# B&R Automation Studio project Template
Automation Studio 4.9

## Logical view

### axisConfiguration.typ - Global data types
```iecst
TYPE
	global_command_typ : 	STRUCT  (*command structure for global commands*)
		Power : BOOL; (*switch on the controller of all axes*)
		Home : BOOL; (*reference all axes*)
		Stop : BOOL; (*stop everey active movement as long as is set (emergency stop)*)
		ErrorAcknowledge : BOOL; (*reset active errors*)
	END_STRUCT;
	psm_command_typ : 	STRUCT  (*command structure for power supply modules*)
		Power : BOOL; (*switch on the controller of the psm*)
		StartPowerMeter : BOOL; (*start the power evaluation of psm*)
		StopPowerMeter : BOOL; (*stop the power evaluation of psm*)
		RestartInterval : BOOL; (*restart the interval of power evaluation*)
	END_STRUCT;
	axis_command_typ : 	STRUCT  (*command structure for single and master axes*)
		Power : BOOL; (*switch on the controller*)
		Home : BOOL; (*reference axis*)
		MoveJogPos : BOOL; (*move in positive direction as long as is set*)
		MoveJogNeg : BOOL; (*move in negative direction as long as is set*)
		MoveAbsolute : BOOL; (*move to a defined position*)
		MoveAdditive : BOOL; (*move a defined distance*)
		MoveVelocity : BOOL; (*start a movement with a defined velocity*)
		Stop : BOOL; (*stop every active movement on the axis as long as is set*)
		Halt : BOOL; (*stop every active movement on the axis*)
	END_STRUCT;
	slave_command_typ : 	STRUCT  (*command structure for slave axes*)
		Power : BOOL; (*switch on the controller*)
		Home : BOOL; (*reference axis*)
		MoveJogPos : BOOL; (*move in positive direction as long as is set*)
		MoveJogNeg : BOOL; (*move in negative direction as long as is set*)
		MoveAbsolute : BOOL; (*move to a defined position*)
		MoveAdditive : BOOL; (*move a defined distance*)
		MoveVelocity : BOOL; (*start a movement with a defined velocity*)
		Stop : BOOL; (*stop every active movement on the axis as long as is set*)
		Halt : BOOL; (*stop every active movement on the axis*)
		StartAutomat : BOOL; (*start coupling between master and slave*)
		StopSlave : BOOL; (*stop coupling between master and slave (automat is still active)*)
		RestartAutomat : BOOL; (*reengage the coupling between master and slave*)
		EndAutomat : BOOL; (*terminate the automat*)
		SetSignal1 : BOOL; (*set the first signal of the automat*)
		SetSignal2 : BOOL; (*set the second signal of the automat*)
		SetSignal3 : BOOL; (*set the third signal of the automat*)
		SetSignal4 : BOOL; (*set the fourth signal of the automat*)
		ResetSignal1 : BOOL; (*reset the first signal of the automat*)
		ResetSignal2 : BOOL; (*reset the second signal of the automat*)
		ResetSignal3 : BOOL; (*reset the third signal of the automat*)
		ResetSignal4 : BOOL; (*reset the fourth signal of the automat*)
	END_STRUCT;
	parameter_typ : 	STRUCT  (*parameter structure*)
		Position : REAL; (*target position for MoveAbsolute-Command*)
		Distance : REAL; (*distance for MoveAdditive-Command*)
		Velocity : REAL; (*velocity for MoveVelocity-Command*)
		Direction : USINT; (*direction for commanded movements*)
		Acceleration : REAL; (*acceleration for commanded movements*)
		Deceleration : REAL; (*deceleration for commanded movements*)
		HomePosition : REAL; (*target position for referencing the axis*)
		HomeMode : USINT; (*homing mode*)
		JogVelocity : REAL; (*velocity for jogging movement*)
	END_STRUCT;
	psm_parameter_typ : 	STRUCT  (*parameter structure for psm*)
		IntervalTime : UINT; (*interval time for the power evaluation*)
	END_STRUCT;
	status_typ : 	STRUCT  (*status structure*)
		ActPosition : REAL; (*actual position of the axis*)
		ActVelocity : REAL; (*actual velocity of the axis*)
		DriveStatus : MC_DRIVESTATUS_TYP; (*actual status of the axis*)
	END_STRUCT;
	slave_status_typ : 	STRUCT  (*status structure*)
		ActPosition : REAL; (*actual position of the axis*)
		ActVelocity : REAL; (*actual velocity of the axis*)
		AutomatRunning : BOOL; (*if set, automat is running*)
		AutomatStandBy : BOOL; (*if set, automat is in stand by*)
		ActualStateIndex : USINT; (*actual state index of the cam automat*)
		ActualStateCamIndex : UINT; (*actual index of the cam profile*)
		InCam : BOOL; (*if set, the cam profile is active*)
		InCompensation : BOOL; (*if set, compensation is active*)
		DriveStatus : MC_DRIVESTATUS_TYP; (*actual status of the axis*)
	END_STRUCT;
	psm_status_typ : 	STRUCT  (*status structure for psm*)
		PowerData : MC_POWERDATA_REF; (*evaluated power data*)
		MissedInterval : UINT; (*MissedIntervals with power evaluation*)
		DriveStatus : MC_DRIVESTATUS_TYP; (*actual status of the axis*)
	END_STRUCT;
	axisState_typ : 	STRUCT  (*axis state structure*)
		Disabled : BOOL; (*if set, axis is in state Disabled*)
		StandStill : BOOL; (*if set, axis is in state StandsStill*)
		Homing : BOOL; (*if set, axis is in state Homing*)
		Stopping : BOOL; (*if set, axis is in state Stopping*)
		DiscreteMotion : BOOL; (*if set, axis is in state DiscreteMotion*)
		ContinuousMotion : BOOL; (*if set, axis is in state ContinuousMotion*)
		SynchronizedMotion : BOOL; (*if set, axis is in state SynchronizedMotion*)
		ErrorStop : BOOL; (*if set, axis is in state ErrorStop*)
	END_STRUCT;
	error_typ : 	STRUCT  (*error structure *)
		AxisErrorCount : UINT; (*number of active axis errors*)
		AxisWarningCount : UINT; (*number of active axis warinings*)
		FunctionBlockErrorCount : UINT; (*number of active function block errors*)
		ErrorRecord : MC_ERRORRECORD_REF; (*error record information*)
		ErrorText : ARRAY[0..3] OF STRING[79]; (*description of first active error or warning*)
	END_STRUCT;
	axis_typ : 	STRUCT  (*substructure for single and master axes*)
		Command : axis_command_typ; (*command structure for single and master axes*)
		Parameter : parameter_typ; (*parameter structure*)
		Status : status_typ; (*status structure*)
		AxisState : axisState_typ; (*axis state structure*)
		Error : error_typ; (*error structure*)
	END_STRUCT;
	slave_typ : 	STRUCT  (*substructure for slave axis*)
		Command : slave_command_typ; (*command structure for slave axes*)
		Parameter : parameter_typ; (*parameter structure*)
		Status : slave_status_typ; (*status structure*)
		AxisState : axisState_typ; (*axis state structure*)
		Error : error_typ; (*error structure*)
	END_STRUCT;
	psm_typ : 	STRUCT  (*substructure for psm*)
		Command : psm_command_typ; (*command structure for psm*)
		Parameter : psm_parameter_typ; (*parameter structure for psm*)
		Status : psm_status_typ; (*status structure for psm*)
		AxisState : axisState_typ; (*axis state structure*)
		Error : error_typ; (*error structure*)
	END_STRUCT;
	global_error_typ : 	STRUCT  (*error structure for global errors*)
		AxisTyp : STRING[10]; (*axis type (Axis, Master or Slave)*)
		AxisIndex : USINT; (*index of error reporting axis (total axis index)*)
		ErrorText : ARRAY[0..3] OF STRING[79]; (*description of first active error or warning*)
		ErrorRecord : MC_ERRORRECORD_REF; (*error record information*)
	END_STRUCT;
END_TYPE
```

### axisConfiguration.var - Global variables
```iecst
VAR CONSTANT
	PSM_NUMBER : USINT := 1; (*number of used power supply modules*)
	AXIS_NUMBER : USINT := 2; (*number of used single axes*)
	MASTER_NUMBER : USINT := 1; (*number of used master axes*)
	SLAVE_NUMBER : USINT := 1; (*number of used slave axes*)
	TOTAL_AXES : USINT := PSM_NUMBER + AXIS_NUMBER + MASTER_NUMBER + SLAVE_NUMBER; (*total number of used axes*)
	PSM_MAX_INDEX : USINT := PSM_NUMBER-1; (*highest index for single axis*)
	AXIS_MAX_INDEX : USINT := AXIS_NUMBER-1; (*highest index for single axes*)
	MASTER_MAX_INDEX : USINT := MASTER_NUMBER-1; (*highest index for master axes*)
	SLAVE_MAX_INDEX : USINT := SLAVE_NUMBER-1; (*highest index for slave axes*)
END_VAR
VAR
	PsmRef : ARRAY[0..PSM_MAX_INDEX] OF UDINT; (*psm reference handle*)
	AxisRef : ARRAY[0..AXIS_MAX_INDEX] OF UDINT; (*axis reference handle*)
	MasterRef : ARRAY[0..MASTER_MAX_INDEX] OF UDINT; (*master reference handle*)
	SlaveRef : ARRAY[0..SLAVE_MAX_INDEX] OF UDINT; (*slave reference handle*)
	GlobalCommand : global_command_typ; (*command structure for global command*)
	GlobalError : global_error_typ; (*error structure for global error*)
	PowerSupply : ARRAY[0..PSM_MAX_INDEX] OF psm_typ; (*handling structure for power supply module*)
	Axis : ARRAY[0..AXIS_MAX_INDEX] OF axis_typ; (*handling structure for single axis*)
	Master : ARRAY[0..MASTER_MAX_INDEX] OF axis_typ; (*handling structure for master axis*)
	Slave : ARRAY[0..SLAVE_MAX_INDEX] OF slave_typ; (*handling structure for slave axis*)
	PowerSupplyOn : BOOL; (*power supply on flag*)
END_VAR
```

### Program Logical/LibACP10MC_MotionControl_ST/AxisConfiguration (IEC) - configuration task

#### axisConfiguration.st - Implementation code
```iecst
(********************************************************************
 * COPYRIGHT -- Bernecker + Rainer
 ********************************************************************
 * Program: AxisConfiguration
 * File: axisConfiguration.st
 * Author: Bernecker + Rainer
 * Created: March 01, 2011
 ********************************************************************
 * Implementation of program AxisConfiguration
 ********************************************************************)

PROGRAM _INIT
    PsmRef[0] := ADR(gAxis01); (* axis reference of the power supply module *)
    AxisRef[0] := ADR(gAxis02); (* axis reference of first single axis *)
    AxisRef[1] := ADR(gAxis03); (* axis reference of second single axis *)
    MasterRef[0] := ADR(gAxis04); (* axis reference of first master axis *)
    SlaveRef[0] := ADR(gAxis05); (* axis reference of first slave axis *)

    PowerSupplyOn := TRUE; (* if a power supply is used, this variable is reset in the according task *)
END_PROGRAM
```

### Program Logical/LibACP10MC_MotionControl_ST/PowerSupply (IEC) - power supply handle

#### powerSupplyCyclic.st - Cyclic code
```iecst
(********************************************************************
 * COPYRIGHT -- Bernecker + Rainer
 ********************************************************************
 * Program: PowerSupply
 * File: powerSupplyCyclic.st
 * Author: Bernecker + Rainer
 * Created: March 01, 2011
 ********************************************************************
 * Implementation of program PowerSupply
 ********************************************************************)

PROGRAM _CYCLIC

(************************** MC_READSTATUS ***************************)
MC_ReadStatus_0.Enable := NOT(MC_ReadStatus_0.Error);
MC_ReadStatus_0.Axis := PsmRef[PSM_INDEX];
MC_ReadStatus_0();
PowerSupply[PSM_INDEX].AxisState.Disabled := MC_ReadStatus_0.Disabled;
PowerSupply[PSM_INDEX].AxisState.StandStill := MC_ReadStatus_0.StandStill;
PowerSupply[PSM_INDEX].AxisState.Stopping := MC_ReadStatus_0.Stopping;
PowerSupply[PSM_INDEX].AxisState.Homing := MC_ReadStatus_0.Homing;
PowerSupply[PSM_INDEX].AxisState.DiscreteMotion := MC_ReadStatus_0.DiscreteMotion;
PowerSupply[PSM_INDEX].AxisState.ContinuousMotion := MC_ReadStatus_0.ContinuousMotion;
PowerSupply[PSM_INDEX].AxisState.SynchronizedMotion := MC_ReadStatus_0.SynchronizedMotion;
PowerSupply[PSM_INDEX].AxisState.ErrorStop := MC_ReadStatus_0.Errorstop;

(************************* MC_BR_READDRIVESTATUS ********************)
MC_BR_ReadDriveStatus_0.Enable := NOT(MC_BR_ReadDriveStatus_0.Error);
MC_BR_ReadDriveStatus_0.Axis := PsmRef[PSM_INDEX];
MC_BR_ReadDriveStatus_0.AdrDriveStatus := ADR(PowerSupply[PSM_INDEX].Status.DriveStatus);
MC_BR_ReadDriveStatus_0();

CASE PsmStep OF
(********************************* READY ****************************)
    STATE_READY:
        IF (((GlobalCommand.Power = TRUE) OR (PowerSupply[PSM_INDEX].Command.Power = TRUE)) AND
             (MC_Power_0.Status = FALSE)) THEN
            PsmStep := STATE_POWER_ON;
        ELSIF ((GlobalCommand.Power = FALSE) AND (PowerSupply[PSM_INDEX].Command.Power = FALSE) AND
                 (MC_Power_0.Status = TRUE)) THEN
            PsmStep := STATE_POWER_OFF;
        ELSIF (PowerSupply[PSM_INDEX].Command.StartPowerMeter = TRUE) THEN
            PowerSupply[PSM_INDEX].Command.StartPowerMeter := FALSE;
            PsmStep := STATE_START_POWERMETER;
        ELSIF (PowerSupply[PSM_INDEX].Command.StopPowerMeter = TRUE) THEN
            PowerSupply[PSM_INDEX].Command.StopPowerMeter := FALSE;
            PsmStep := STATE_STOP_POWERMETER;
        ELSIF (PowerSupply[PSM_INDEX].Command.RestartInterval = TRUE) THEN
            PowerSupply[PSM_INDEX].Command.RestartInterval := FALSE;
            MC_BR_PowerMeter_0.RestartInterval := FALSE;
            PsmStep := STATE_RESTART_INTERVAL;
        END_IF

        (* End of STATE_READY *)

(*************************** POWER ON ********************************)
    STATE_POWER_ON:
        MC_Power_0.Enable := TRUE;
        IF (MC_Power_0.Status = TRUE) THEN
            PsmStep := STATE_READY;
        END_IF

        (* IF a power error occured switch off controller *)
        IF (MC_Power_0.Error = TRUE) THEN
            MC_Power_0.Enable := FALSE;
        END_IF

        (* End of STATE_POWER_ON *)

(************************* POWER OFF *******************************)
    STATE_POWER_OFF:
        MC_Power_0.Enable := FALSE;
        IF (MC_Power_0.Status = FALSE) THEN
            PsmStep := STATE_READY;
        END_IF

        (* End of STATE_POWER_OFF *)

(************************ START POWERMETER **************************)
    STATE_START_POWERMETER:
        MC_BR_PowerMeter_0.Enable := TRUE;
        MC_BR_PowerMeter_0.Mode := mcONLY_PSM;
        MC_BR_PowerMeter_0.IntervalTime := PowerSupply[PSM_INDEX].Parameter.IntervalTime;

        IF (MC_BR_PowerMeter_0.Valid = TRUE) THEN
            PsmStep := STATE_READY;
        END_IF

        (* check IF error occured *)
        IF (MC_BR_PowerMeter_0.Error = TRUE) THEN
            MC_BR_PowerMeter_0.Enable := FALSE;
            PsmStep := STATE_READY;
        END_IF

        (* End of STATE_START_POWERMETER *)

(************************ STOP POWERMETER ***************************)
    STATE_STOP_POWERMETER:
        MC_BR_PowerMeter_0.Enable := FALSE;

        IF (MC_BR_PowerMeter_0.Valid = FALSE) THEN
            PsmStep := STATE_READY;
        END_IF

        (* End of STATE_STOP_POWERMETER *)

(********************** STATE RESTART INTERVAL **********************)
    STATE_RESTART_INTERVAL:
        MC_BR_PowerMeter_0.RestartInterval := TRUE;
        PsmStep := STATE_READY;

        (* End of STATE_RESTART_INTERVAL *)

(*********************** SEQUENCE END *******************************)
END_CASE

(*********************************************************************
        Function Block Calls
*********************************************************************)

(*************************** MC_POWER *******************************)
MC_Power_0.Axis := PsmRef[PSM_INDEX];
MC_Power_0();
PowerSupplyOn := MC_Power_0.Status;

(**********************MC_BR_POWERMETER *****************************)
MC_BR_PowerMeter_0.Axis := PsmRef[PSM_INDEX];
MC_BR_PowerMeter_0();
PowerSupply[PSM_INDEX].Status.PowerData.IntervalNumber        := MC_BR_PowerMeter_0.PowerData.IntervalNumber;
PowerSupply[PSM_INDEX].Status.PowerData.IntervalDuration      := MC_BR_PowerMeter_0.PowerData.IntervalDuration;
PowerSupply[PSM_INDEX].Status.PowerData.AverageActivePower    := MC_BR_PowerMeter_0.PowerData.AverageActivePower;
PowerSupply[PSM_INDEX].Status.PowerData.AverageReactivePower  := MC_BR_PowerMeter_0.PowerData.AverageReactivePower;
PowerSupply[PSM_INDEX].Status.PowerData.MaximumActivePower    := MC_BR_PowerMeter_0.PowerData.MaximumActivePower;
PowerSupply[PSM_INDEX].Status.PowerData.MinimalActivePower    := MC_BR_PowerMeter_0.PowerData.MinimalActivePower;
PowerSupply[PSM_INDEX].Status.PowerData.ConsumedEnergy        := MC_BR_PowerMeter_0.PowerData.ConsumedEnergy;
PowerSupply[PSM_INDEX].Status.PowerData.RegeneratedEnergy     := MC_BR_PowerMeter_0.PowerData.RegeneratedEnergy;
PowerSupply[PSM_INDEX].Status.PowerData.EnergyBalance         := MC_BR_PowerMeter_0.PowerData.EnergyBalance;

END_PROGRAM
```

#### powerSupplyInit.st - Initialization code
```iecst
(********************************************************************
 * COPYRIGHT -- Bernecker + Rainer
 ********************************************************************
 * Program: PowerSupply
 * File: powerSupplyInit.st
 * Author: Bernecker + Rainer
 * Created: March 01, 2011
 ********************************************************************
 * Implementation of program PowerSupply
 ********************************************************************)

PROGRAM _INIT
PsmStep := STATE_READY;

PowerSupply[PSM_INDEX].Parameter.IntervalTime := 10000; (* IntervalTime of 10sec *)
END_PROGRAM
```

#### powerSupply.var - Local variables
```iecst
VAR CONSTANT
	PSM_INDEX : USINT := 0;
	STATE_READY : USINT := 0;
	STATE_POWER_ON : USINT := 1;
	STATE_POWER_OFF : USINT := 2;
	STATE_START_POWERMETER : USINT := 3;
	STATE_STOP_POWERMETER : USINT := 4;
	STATE_RESTART_INTERVAL : USINT := 5;
END_VAR
VAR
	MC_Power_0 : MC_Power;
	MC_BR_PowerMeter_0 : MC_BR_PowerMeter;
	MC_BR_ReadDriveStatus_0 : MC_BR_ReadDriveStatus;
	MC_ReadStatus_0 : MC_ReadStatus;
	PsmStep : USINT;
END_VAR
```

### Program Logical/LibACP10MC_MotionControl_ST/Axis_00 (IEC) - single axis handle

#### axisCyclic.st - Cyclic code
```iecst
(********************************************************************
 * COPYRIGHT -- Bernecker + Rainer
 ********************************************************************
 * Program: Axis_00
 * File: axisCyclic.st
 * Author: Bernecker + Rainer
 * Created: March 01, 2011
 ********************************************************************
 * Implementation of program Axis_00
 ********************************************************************)

PROGRAM _CYCLIC

(*********** CHECK IF POWER SHOULD BE OFF ***************************)
    IF ((GlobalCommand.Power = FALSE) AND (Axis[AXIS_INDEX].Command.Power = FALSE)) THEN
        AxisStep := STATE_WAIT;
    END_IF

    (* central monitoring of the stop command allows a shorter reaction time *)
    IF ((GlobalCommand.Stop = TRUE) OR (Axis[AXIS_INDEX].Command.Stop = TRUE)) THEN
        IF ((GlobalCommand.Power = TRUE) OR (Axis[AXIS_INDEX].Command.Power = TRUE)) THEN
            AxisStep := STATE_STOP;
            (* reset all FB execute inputs we use *)
            MC_Home_0.Execute := FALSE;
            MC_Halt_0.Execute := FALSE;
            MC_MoveAbsolute_0.Execute := FALSE;
            MC_MoveAdditive_0.Execute := FALSE;
            MC_MoveVelocity_0.Execute := FALSE;

            Axis[AXIS_INDEX].Command.MoveJogPos := FALSE;
            Axis[AXIS_INDEX].Command.MoveJogNeg := FALSE;
        END_IF
    END_IF

(************************** MC_READSTATUS ***************************)
MC_ReadStatus_0.Enable := NOT(MC_ReadStatus_0.Error);
MC_ReadStatus_0.Axis := AxisRef[AXIS_INDEX];
MC_ReadStatus_0();
Axis[AXIS_INDEX].AxisState.Disabled             := MC_ReadStatus_0.Disabled;
Axis[AXIS_INDEX].AxisState.StandStill           := MC_ReadStatus_0.StandStill;
Axis[AXIS_INDEX].AxisState.Stopping             := MC_ReadStatus_0.Stopping;
Axis[AXIS_INDEX].AxisState.Homing               := MC_ReadStatus_0.Homing;
Axis[AXIS_INDEX].AxisState.DiscreteMotion       := MC_ReadStatus_0.DiscreteMotion;
Axis[AXIS_INDEX].AxisState.ContinuousMotion     := MC_ReadStatus_0.ContinuousMotion;
Axis[AXIS_INDEX].AxisState.SynchronizedMotion   := MC_ReadStatus_0.SynchronizedMotion;
Axis[AXIS_INDEX].AxisState.ErrorStop            := MC_ReadStatus_0.Errorstop;

(********************** MC_BR_READDRIVESTATUS ***********************)
MC_BR_ReadDriveStatus_0.Enable := NOT(MC_BR_ReadDriveStatus_0.Error);
MC_BR_ReadDriveStatus_0.Axis := AxisRef[AXIS_INDEX];
MC_BR_ReadDriveStatus_0.AdrDriveStatus := ADR(Axis[AXIS_INDEX].Status.DriveStatus);
MC_BR_ReadDriveStatus_0();

(********************* MC_READACTUALPOSITION ************************)
MC_ReadActualPosition_0.Enable := NOT(MC_ReadActualPosition_0.Error);
MC_ReadActualPosition_0.Axis := AxisRef[AXIS_INDEX];
MC_ReadActualPosition_0();
IF(MC_ReadActualPosition_0.Valid = TRUE) THEN
    Axis[AXIS_INDEX].Status.ActPosition := MC_ReadActualPosition_0.Position;
END_IF

(********************* MC_READACTUALVELOCITY ************************)
MC_ReadActualVelocity_0.Enable := NOT(MC_ReadActualVelocity_0.Error);
MC_ReadActualVelocity_0.Axis := AxisRef[AXIS_INDEX];
MC_ReadActualVelocity_0();
IF(MC_ReadActualVelocity_0.Valid = TRUE) THEN
    Axis[AXIS_INDEX].Status.ActVelocity := MC_ReadActualVelocity_0.Velocity;
END_IF

CASE AxisStep OF
(****************************** WAIT ********************************)
    STATE_WAIT: (* STATE: Wait *)
        IF ((GlobalCommand.Power = TRUE) OR (Axis[AXIS_INDEX].Command.Power = TRUE)) THEN
            AxisStep := STATE_POWER_ON;
        ELSE
            MC_Power_0.Enable := FALSE;
        END_IF

        (* reset all FB execute inputs we use *)
        MC_Home_0.Execute := FALSE;
        MC_Halt_0.Execute := FALSE;
        MC_Stop_0.Execute := FALSE;
        MC_MoveAbsolute_0.Execute := FALSE;
        MC_MoveAdditive_0.Execute := FALSE;
        MC_MoveVelocity_0.Execute := FALSE;

        (* reset user commands *)
        Axis[AXIS_INDEX].Command.Stop := FALSE;
        Axis[AXIS_INDEX].Command.MoveJogPos := FALSE;
        Axis[AXIS_INDEX].Command.MoveJogNeg := FALSE;
        Axis[AXIS_INDEX].Command.MoveVelocity := FALSE;
        Axis[AXIS_INDEX].Command.MoveAbsolute := FALSE;
        Axis[AXIS_INDEX].Command.MoveAdditive := FALSE;

    (* End of STATE_WAIT *)

(****************************** POWER ON ****************************)
    STATE_POWER_ON: (* STATE: Power on *)
        IF (PowerSupplyOn = TRUE) THEN
            MC_Power_0.Enable := TRUE;
        END_IF
        IF (MC_Power_0.Status = TRUE) THEN
            AxisStep := STATE_READY;
        END_IF

        (* if a power error occured switch off controller *)
        IF (MC_Power_0.Error = TRUE) THEN
            MC_Power_0.Enable := FALSE;
        END_IF

        (* End of STATE_POWER_ON *)

(****************************** READY *******************************)
    STATE_READY: (* STATE: Waiting for Commands *)
        IF ((Axis[AXIS_INDEX].Command.Home = TRUE) OR (GlobalCommand.Home = TRUE)) THEN
            Axis[AXIS_INDEX].Command.Home := FALSE;
            AxisStep := STATE_HOME;
        ELSIF ((Axis[AXIS_INDEX].Command.Stop = TRUE) OR (GlobalCommand.Stop = TRUE)) THEN
            AxisStep := STATE_STOP;
        ELSIF (Axis[AXIS_INDEX].Command.MoveJogPos = TRUE) THEN
            AxisStep := STATE_JOG_POSITIVE;
        ELSIF (Axis[AXIS_INDEX].Command.MoveJogNeg = TRUE) THEN
            AxisStep := STATE_JOG_NEGATIVE;
        ELSIF (Axis[AXIS_INDEX].Command.MoveAbsolute = TRUE) THEN
            Axis[AXIS_INDEX].Command.MoveAbsolute := FALSE;
            AxisStep := STATE_MOVE_ABSOLUTE;
        ELSIF (Axis[AXIS_INDEX].Command.MoveAdditive = TRUE) THEN
            Axis[AXIS_INDEX].Command.MoveAdditive := FALSE;
            AxisStep := STATE_MOVE_ADDITIVE;
        ELSIF (Axis[AXIS_INDEX].Command.MoveVelocity = TRUE) THEN
            Axis[AXIS_INDEX].Command.MoveVelocity := FALSE;
            AxisStep := STATE_MOVE_VELOCITY;
        ELSIF (Axis[AXIS_INDEX].Command.Halt = TRUE) THEN
            Axis[AXIS_INDEX].Command.Halt := FALSE;
            AxisStep := STATE_HALT;
        END_IF

        (* End of STATE_READY *)

(****************************** HOME ********************************)
    STATE_HOME: (* STATE: start homing process *)
        MC_Home_0.Position := Axis[AXIS_INDEX].Parameter.HomePosition;
        MC_Home_0.HomingMode := Axis[AXIS_INDEX].Parameter.HomeMode;
        MC_Home_0.Execute := TRUE;
        IF (MC_Home_0.Done = TRUE) THEN
            GlobalCommand.Home := FALSE;
            MC_Home_0.Execute := FALSE;
            AxisStep := STATE_READY;
        END_IF

        (* if a homing error occured go to ready state *)
        IF ((MC_Home_0.Error = TRUE) OR (MC_Home_0.CommandAborted = TRUE)) THEN
            MC_Home_0.Execute := FALSE;
            AxisStep := STATE_READY;
        END_IF

        (* End of STATE_HOME *)

(*************************** HALT MOVEMENT **************************)
    STATE_HALT: (* STATE: Stop the active movement *)
        MC_Halt_0.Deceleration := Axis[AXIS_INDEX].Parameter.Deceleration;
        MC_Halt_0.Execute := TRUE;
        IF (MC_Halt_0.Done = TRUE) THEN
            MC_Halt_0.Execute := FALSE;
            AxisStep := STATE_READY;
       END_IF

       (* check if error occured *)
       IF ((MC_Halt_0.Error = TRUE) OR (MC_Halt_0.CommandAborted = TRUE)) THEN
           MC_Halt_0.Execute := FALSE;
           AxisStep := STATE_READY;
       END_IF

       (* End of STATE_HALT *)

(*************************** STOP MOVEMENT **************************)
    STATE_STOP: (* STATE: Stop movement as long as command is set *)
        MC_Stop_0.Deceleration := Axis[AXIS_INDEX].Parameter.Deceleration;
        MC_Stop_0.Execute := TRUE;

        (* if axis is stopped go to ready state *)
        IF ((MC_Stop_0.Done = TRUE) AND (Axis[AXIS_INDEX].Command.Stop = FALSE) AND (GlobalCommand.Stop = FALSE)) THEN
            MC_Stop_0.Execute := FALSE;
            AxisStep := STATE_READY;
        END_IF

        (* check if error occured *)
        IF (((MC_Stop_0.Error = TRUE) OR (MC_Stop_0.CommandAborted = TRUE)) AND
             (Axis[AXIS_INDEX].Command.Stop = FALSE) AND
             (GlobalCommand.Stop = FALSE)) THEN
            MC_Stop_0.Execute := FALSE;
            AxisStep := STATE_READY;
        END_IF

       (* End of STATE_STOP *)

(******************* START JOG MOVEMENT POSITIVE ********************)
    STATE_JOG_POSITIVE: (* STATE: Start jog movement in positive direction *)
        MC_MoveVelocity_0.Velocity      := Axis[AXIS_INDEX].Parameter.JogVelocity;
        MC_MoveVelocity_0.Acceleration  := Axis[AXIS_INDEX].Parameter.Acceleration;
        MC_MoveVelocity_0.Deceleration  := Axis[AXIS_INDEX].Parameter.Deceleration;
        MC_MoveVelocity_0.Direction     := mcPOSITIVE_DIR;
        MC_MoveVelocity_0.Execute := 1;

        (* check if jog movement should be stopped *)
        IF (Axis[AXIS_INDEX].Command.MoveJogPos = FALSE) THEN
            MC_MoveVelocity_0.Execute := FALSE;
            AxisStep := STATE_HALT;
        END_IF

        IF ((MC_MoveVelocity_0.Error = TRUE) OR (MC_MoveVelocity_0.CommandAborted = TRUE)) THEN
            MC_MoveVelocity_0.Execute := FALSE;
            AxisStep := STATE_READY;
        END_IF

        (* End of STATE_JOG_POSITIVE *)

(********************START JOG MOVEMENT NEGATIVE ********************)
    STATE_JOG_NEGATIVE: (* STATE: Start jog movement in negative direction *)
        MC_MoveVelocity_0.Velocity      := Axis[AXIS_INDEX].Parameter.JogVelocity;
        MC_MoveVelocity_0.Acceleration  := Axis[AXIS_INDEX].Parameter.Acceleration;
        MC_MoveVelocity_0.Deceleration  := Axis[AXIS_INDEX].Parameter.Deceleration;
        MC_MoveVelocity_0.Direction     := mcNEGATIVE_DIR;
        MC_MoveVelocity_0.Execute := 1;

        (* check if jog movement should be stopped *)
        IF (Axis[AXIS_INDEX].Command.MoveJogNeg = FALSE) THEN
            MC_MoveVelocity_0.Execute := FALSE;
            AxisStep := STATE_HALT;
        END_IF

        IF ((MC_MoveVelocity_0.Error = TRUE) OR (MC_MoveVelocity_0.CommandAborted = TRUE)) THEN
            MC_MoveVelocity_0.Execute := FALSE;
            AxisStep := STATE_READY;
        END_IF

        (* End of STATE_JOG_NEGATIVE *)

(********************* START ABSOLUTE MOVEMENT **********************)
    STATE_MOVE_ABSOLUTE: (* STATE: Start absolute movement *)
        MC_MoveAbsolute_0.Position      := Axis[AXIS_INDEX].Parameter.Position;
        MC_MoveAbsolute_0.Velocity      := Axis[AXIS_INDEX].Parameter.Velocity;
        MC_MoveAbsolute_0.Acceleration  := Axis[AXIS_INDEX].Parameter.Acceleration;
        MC_MoveAbsolute_0.Deceleration  := Axis[AXIS_INDEX].Parameter.Deceleration;
        MC_MoveAbsolute_0.Direction     := Axis[AXIS_INDEX].Parameter.Direction;
        MC_MoveAbsolute_0.Execute := 1;

        IF (Axis[AXIS_INDEX].Command.Halt = TRUE) THEN
            Axis[AXIS_INDEX].Command.Halt := 0;
            MC_MoveAbsolute_0.Execute := 0;
            AxisStep := STATE_HALT;
        ELSIF (MC_MoveAbsolute_0.Done = TRUE) THEN
            MC_MoveAbsolute_0.Execute := FALSE;
            AxisStep := STATE_READY;
        END_IF

        IF ((MC_MoveAbsolute_0.Error = TRUE) OR (MC_MoveAbsolute_0.CommandAborted = TRUE)) THEN
            MC_MoveAbsolute_0.Execute := FALSE;
            AxisStep := STATE_READY;
        END_IF

        (* End of STATE_MOVE_ABSOLUTE *)

(********************* START ADDITIVE MOVEMENT **********************)
    STATE_MOVE_ADDITIVE: (* STATE: Start additive movement *)
        MC_MoveAdditive_0.Distance      := Axis[AXIS_INDEX].Parameter.Distance;
        MC_MoveAdditive_0.Velocity      := Axis[AXIS_INDEX].Parameter.Velocity;
        MC_MoveAdditive_0.Acceleration  := Axis[AXIS_INDEX].Parameter.Acceleration;
        MC_MoveAdditive_0.Deceleration  := Axis[AXIS_INDEX].Parameter.Deceleration;
        MC_MoveAdditive_0.Execute := 1;
        IF (Axis[AXIS_INDEX].Command.Halt = TRUE) THEN
            Axis[AXIS_INDEX].Command.Halt := FALSE;
            MC_MoveAdditive_0.Execute := FALSE;
            AxisStep := STATE_HALT;
        ELSIF (MC_MoveAdditive_0.Done = TRUE) THEN
            MC_MoveAdditive_0.Execute := FALSE;
             AxisStep := STATE_READY;
        END_IF

        (* check IF error occured *)
        IF ((MC_MoveAdditive_0.Error = TRUE) OR (MC_MoveAdditive_0.CommandAborted = TRUE)) THEN
            MC_MoveAdditive_0.Execute := FALSE;
            AxisStep := STATE_READY;
        END_IF

        (* End of STATE_MOVE_ADDITIVE *)

(********************* START VELOCITY MOVEMENT **********************)
    STATE_MOVE_VELOCITY: (* STATE: Start velocity movement *)
        MC_MoveVelocity_0.Velocity      := Axis[AXIS_INDEX].Parameter.Velocity;
        MC_MoveVelocity_0.Acceleration  := Axis[AXIS_INDEX].Parameter.Acceleration;
        MC_MoveVelocity_0.Deceleration  := Axis[AXIS_INDEX].Parameter.Deceleration;
        MC_MoveVelocity_0.Direction     := Axis[AXIS_INDEX].Parameter.Direction;
        MC_MoveVelocity_0.Execute := 1;

        IF (Axis[AXIS_INDEX].Command.Halt = TRUE) THEN
            Axis[AXIS_INDEX].Command.Halt := FALSE;
            MC_MoveVelocity_0.Execute := FALSE;
            AxisStep := STATE_HALT;
        ELSIF (MC_MoveVelocity_0.InVelocity = TRUE) THEN
            MC_MoveVelocity_0.Execute := FALSE;
             AxisStep := STATE_READY;
        END_IF
        (* check if error occured *)
        IF ((MC_MoveVelocity_0.Error = TRUE) OR (MC_MoveVelocity_0.CommandAborted = TRUE)) THEN
            MC_MoveVelocity_0.Execute := FALSE;
            AxisStep := STATE_READY;
        END_IF

        (* End of STATE_MOVE_ADDITIVE *)

(*********************** SEQUENCE END *******************************)
END_CASE

(*********************************************************************
        Function Block Calls
*********************************************************************)

(*************************** MC_POWER *******************************)
MC_Power_0.Axis := AxisRef[AXIS_INDEX];
MC_Power_0();

(**************************** MC_HOME *******************************)
MC_Home_0.Axis := AxisRef[AXIS_INDEX];
MC_Home_0();

(************************ MC_MOVEABSOLUTE ***************************)
MC_MoveAbsolute_0.Axis := AxisRef[AXIS_INDEX];
MC_MoveAbsolute_0();

(************************ MC_MOVEADDITIVE ***************************)
MC_MoveAdditive_0.Axis := AxisRef[AXIS_INDEX];
MC_MoveAdditive_0();

(************************ MC_MOVEVELOCITY ***************************)
MC_MoveVelocity_0.Axis := AxisRef[AXIS_INDEX];
MC_MoveVelocity_0();

(**************************** MC_STOP *******************************)
MC_Stop_0.Axis := AxisRef[AXIS_INDEX];
MC_Stop_0();

(****************************MC_HALT*********************************)
MC_Halt_0.Axis := AxisRef[AXIS_INDEX];
MC_Halt_0();

END_PROGRAM
```

#### axisInit.st - Initialization code
```iecst
(********************************************************************
 * COPYRIGHT -- Bernecker + Rainer
 ********************************************************************
 * Program: Axis_00
 * File: axisInit.st
 * Author: Bernecker + Rainer
 * Created: March 01, 2011
 ********************************************************************
 * Implementation of program Axis_00
 ********************************************************************)

PROGRAM _INIT
AxisStep := STATE_WAIT; (* start step *)

Axis[AXIS_INDEX].Parameter.Velocity       := 1000; (* velocity for movement *)
Axis[AXIS_INDEX].Parameter.Acceleration   := 5000; (* acceleration for movement *)
Axis[AXIS_INDEX].Parameter.Deceleration   := 5000; (* deceleration for movement *)
Axis[AXIS_INDEX].Parameter.JogVelocity    := 400;  (* velocity for jogging *)
END_PROGRAM
```

#### axis.var - Local variables
```iecst
(*Actual step inside the step sequencer*)
VAR
	AxisStep : USINT; (*current step in the step sequence*)
END_VAR
VAR CONSTANT
	STATE_WAIT : USINT := 0; (*constant for a waiting step*)
	STATE_POWER_ON : USINT := 1; (*constant for the step in which the controller is switched on*)
	STATE_HOME : USINT := 2; (*constant for the step in which the axis is referenced*)
	STATE_READY : USINT := 10; (*constant for a waiting step*)
	STATE_HALT : USINT := 11; (*constant for the step in which movements are stopped*)
	STATE_STOP : USINT := 12; (*constant for the step in which movements are stopped *)
	STATE_JOG_POSITIVE : USINT := 13; (*constant for the step in which positive jogging movement is executed*)
	STATE_JOG_NEGATIVE : USINT := 14; (*constant for the step in which negative jogging movement is executed*)
	STATE_MOVE_ABSOLUTE : USINT := 15; (*constant for the step in which a movement to defined position is executed*)
	STATE_MOVE_ADDITIVE : USINT := 16; (*constant for the step in which a movement with defined distance is executed*)
	STATE_MOVE_VELOCITY : USINT := 17; (*constant for the step in which a movement with defined velocity is started*)
END_VAR
(*Index of the used axis*)
VAR CONSTANT
	AXIS_INDEX : USINT := 0; (*Index of the used axis*)
END_VAR
(*Function Blocks*)
VAR
	MC_BR_ReadDriveStatus_0 : MC_BR_ReadDriveStatus; (*Function Block*)
	MC_Halt_0 : MC_Halt; (*Function Block*)
	MC_Home_0 : MC_Home; (*Function Block*)
	MC_MoveAbsolute_0 : MC_MoveAbsolute; (*Function Block*)
	MC_MoveAdditive_0 : MC_MoveAdditive; (*Function Block*)
	MC_MoveVelocity_0 : MC_MoveVelocity; (*Function Block*)
	MC_Power_0 : MC_Power; (*Function Block*)
	MC_ReadActualPosition_0 : MC_ReadActualPosition; (*Function Block*)
	MC_ReadActualVelocity_0 : MC_ReadActualVelocity; (*Function Block*)
	MC_ReadStatus_0 : MC_ReadStatus; (*Function Block*)
	MC_Stop_0 : MC_Stop; (*Function Block*)
END_VAR
```

### Program Logical/LibACP10MC_MotionControl_ST/Axis_01 (IEC) - single axis handle

#### axisCyclic.st
```iecst
(********************************************************************
 * COPYRIGHT -- Bernecker + Rainer
 ********************************************************************
 * Program: Axis_00
 * File: axisCyclic.st
 * Author: Bernecker + Rainer
 * Created: March 01, 2011
 ********************************************************************
 * Implementation of program Axis_00
 ********************************************************************)

PROGRAM _CYCLIC

(*********** CHECK IF POWER SHOULD BE OFF ***************************)
    IF ((GlobalCommand.Power = FALSE) AND (Axis[AXIS_INDEX].Command.Power = FALSE)) THEN
        AxisStep := STATE_WAIT;
    END_IF

    (* central monitoring of the stop command allows a shorter reaction time *)
    IF ((GlobalCommand.Stop = TRUE) OR (Axis[AXIS_INDEX].Command.Stop = TRUE)) THEN
        IF ((GlobalCommand.Power = TRUE) OR (Axis[AXIS_INDEX].Command.Power = TRUE)) THEN
            AxisStep := STATE_STOP;
            (* reset all FB execute inputs we use *)
            MC_Home_0.Execute := FALSE;
            MC_Halt_0.Execute := FALSE;
            MC_MoveAbsolute_0.Execute := FALSE;
            MC_MoveAdditive_0.Execute := FALSE;
            MC_MoveVelocity_0.Execute := FALSE;

            Axis[AXIS_INDEX].Command.MoveJogPos := FALSE;
            Axis[AXIS_INDEX].Command.MoveJogNeg := FALSE;
        END_IF
    END_IF

(************************** MC_READSTATUS ***************************)
MC_ReadStatus_0.Enable := NOT(MC_ReadStatus_0.Error);
MC_ReadStatus_0.Axis := AxisRef[AXIS_INDEX];
MC_ReadStatus_0();
Axis[AXIS_INDEX].AxisState.Disabled             := MC_ReadStatus_0.Disabled;
Axis[AXIS_INDEX].AxisState.StandStill           := MC_ReadStatus_0.StandStill;
Axis[AXIS_INDEX].AxisState.Stopping             := MC_ReadStatus_0.Stopping;
Axis[AXIS_INDEX].AxisState.Homing               := MC_ReadStatus_0.Homing;
Axis[AXIS_INDEX].AxisState.DiscreteMotion       := MC_ReadStatus_0.DiscreteMotion;
Axis[AXIS_INDEX].AxisState.ContinuousMotion     := MC_ReadStatus_0.ContinuousMotion;
Axis[AXIS_INDEX].AxisState.SynchronizedMotion   := MC_ReadStatus_0.SynchronizedMotion;
Axis[AXIS_INDEX].AxisState.ErrorStop            := MC_ReadStatus_0.Errorstop;

(********************** MC_BR_READDRIVESTATUS ***********************)
MC_BR_ReadDriveStatus_0.Enable := NOT(MC_BR_ReadDriveStatus_0.Error);
MC_BR_ReadDriveStatus_0.Axis := AxisRef[AXIS_INDEX];
MC_BR_ReadDriveStatus_0.AdrDriveStatus := ADR(Axis[AXIS_INDEX].Status.DriveStatus);
MC_BR_ReadDriveStatus_0();

(********************* MC_READACTUALPOSITION ************************)
MC_ReadActualPosition_0.Enable := NOT(MC_ReadActualPosition_0.Error);
MC_ReadActualPosition_0.Axis := AxisRef[AXIS_INDEX];
MC_ReadActualPosition_0();
IF(MC_ReadActualPosition_0.Valid = TRUE) THEN
    Axis[AXIS_INDEX].Status.ActPosition := MC_ReadActualPosition_0.Position;
END_IF

(********************* MC_READACTUALVELOCITY ************************)
MC_ReadActualVelocity_0.Enable := NOT(MC_ReadActualVelocity_0.Error);
MC_ReadActualVelocity_0.Axis := AxisRef[AXIS_INDEX];
MC_ReadActualVelocity_0();
IF(MC_ReadActualVelocity_0.Valid = TRUE) THEN
    Axis[AXIS_INDEX].Status.ActVelocity := MC_ReadActualVelocity_0.Velocity;
END_IF

CASE AxisStep OF
(****************************** WAIT ********************************)
    STATE_WAIT: (* STATE: Wait *)
        IF ((GlobalCommand.Power = TRUE) OR (Axis[AXIS_INDEX].Command.Power = TRUE)) THEN
            AxisStep := STATE_POWER_ON;
        ELSE
            MC_Power_0.Enable := FALSE;
        END_IF

        (* reset all FB execute inputs we use *)
        MC_Home_0.Execute := FALSE;
        MC_Halt_0.Execute := FALSE;
        MC_Stop_0.Execute := FALSE;
        MC_MoveAbsolute_0.Execute := FALSE;
        MC_MoveAdditive_0.Execute := FALSE;
        MC_MoveVelocity_0.Execute := FALSE;

        (* reset user commands *)
        Axis[AXIS_INDEX].Command.Stop := FALSE;
        Axis[AXIS_INDEX].Command.MoveJogPos := FALSE;
        Axis[AXIS_INDEX].Command.MoveJogNeg := FALSE;
        Axis[AXIS_INDEX].Command.MoveVelocity := FALSE;
        Axis[AXIS_INDEX].Command.MoveAbsolute := FALSE;
        Axis[AXIS_INDEX].Command.MoveAdditive := FALSE;

    (* End of STATE_WAIT *)

(****************************** POWER ON ****************************)
    STATE_POWER_ON: (* STATE: Power on *)
        IF (PowerSupplyOn = TRUE) THEN
            MC_Power_0.Enable := TRUE;
        END_IF
        IF (MC_Power_0.Status = TRUE) THEN
            AxisStep := STATE_READY;
        END_IF

        (* if a power error occured switch off controller *)
        IF (MC_Power_0.Error = TRUE) THEN
            MC_Power_0.Enable := FALSE;
        END_IF

        (* End of STATE_POWER_ON *)

(****************************** READY *******************************)
    STATE_READY: (* STATE: Waiting for Commands *)
        IF ((Axis[AXIS_INDEX].Command.Home = TRUE) OR (GlobalCommand.Home = TRUE)) THEN
            Axis[AXIS_INDEX].Command.Home := FALSE;
            AxisStep := STATE_HOME;
        ELSIF ((Axis[AXIS_INDEX].Command.Stop = TRUE) OR (GlobalCommand.Stop = TRUE)) THEN
            AxisStep := STATE_STOP;
        ELSIF (Axis[AXIS_INDEX].Command.MoveJogPos = TRUE) THEN
            AxisStep := STATE_JOG_POSITIVE;
        ELSIF (Axis[AXIS_INDEX].Command.MoveJogNeg = TRUE) THEN
            AxisStep := STATE_JOG_NEGATIVE;
        ELSIF (Axis[AXIS_INDEX].Command.MoveAbsolute = TRUE) THEN
            Axis[AXIS_INDEX].Command.MoveAbsolute := FALSE;
            AxisStep := STATE_MOVE_ABSOLUTE;
        ELSIF (Axis[AXIS_INDEX].Command.MoveAdditive = TRUE) THEN
            Axis[AXIS_INDEX].Command.MoveAdditive := FALSE;
            AxisStep := STATE_MOVE_ADDITIVE;
        ELSIF (Axis[AXIS_INDEX].Command.MoveVelocity = TRUE) THEN
            Axis[AXIS_INDEX].Command.MoveVelocity := FALSE;
            AxisStep := STATE_MOVE_VELOCITY;
        ELSIF (Axis[AXIS_INDEX].Command.Halt = TRUE) THEN
            Axis[AXIS_INDEX].Command.Halt := FALSE;
            AxisStep := STATE_HALT;
        END_IF

        (* End of STATE_READY *)

(****************************** HOME ********************************)
    STATE_HOME: (* STATE: start homing process *)
        MC_Home_0.Position := Axis[AXIS_INDEX].Parameter.HomePosition;
        MC_Home_0.HomingMode := Axis[AXIS_INDEX].Parameter.HomeMode;
        MC_Home_0.Execute := TRUE;
        IF (MC_Home_0.Done = TRUE) THEN
            GlobalCommand.Home := FALSE;
            MC_Home_0.Execute := FALSE;
            AxisStep := STATE_READY;
        END_IF

        (* if a homing error occured go to ready state *)
        IF ((MC_Home_0.Error = TRUE) OR (MC_Home_0.CommandAborted = TRUE)) THEN
            MC_Home_0.Execute := FALSE;
            AxisStep := STATE_READY;
        END_IF

        (* End of STATE_HOME *)

(*************************** HALT MOVEMENT **************************)
    STATE_HALT: (* STATE: Stop the active movement *)
        MC_Halt_0.Deceleration := Axis[AXIS_INDEX].Parameter.Deceleration;
        MC_Halt_0.Execute := TRUE;
        IF (MC_Halt_0.Done = TRUE) THEN
            MC_Halt_0.Execute := FALSE;
            AxisStep := STATE_READY;
       END_IF

       (* check if error occured *)
       IF ((MC_Halt_0.Error = TRUE) OR (MC_Halt_0.CommandAborted = TRUE)) THEN
           MC_Halt_0.Execute := FALSE;
           AxisStep := STATE_READY;
       END_IF

       (* End of STATE_HALT *)

(*************************** STOP MOVEMENT **************************)
    STATE_STOP: (* STATE: Stop movement as long as command is set *)
        MC_Stop_0.Deceleration := Axis[AXIS_INDEX].Parameter.Deceleration;
        MC_Stop_0.Execute := TRUE;

        (* if axis is stopped go to ready state *)
        IF ((MC_Stop_0.Done = TRUE) AND (Axis[AXIS_INDEX].Command.Stop = FALSE) AND (GlobalCommand.Stop = FALSE)) THEN
            MC_Stop_0.Execute := FALSE;
            AxisStep := STATE_READY;
        END_IF

        (* check if error occured *)
        IF (((MC_Stop_0.Error = TRUE) OR (MC_Stop_0.CommandAborted = TRUE)) AND
             (Axis[AXIS_INDEX].Command.Stop = FALSE) AND
             (GlobalCommand.Stop = FALSE)) THEN
            MC_Stop_0.Execute := FALSE;
            AxisStep := STATE_READY;
        END_IF

       (* End of STATE_STOP *)

(******************* START JOG MOVEMENT POSITIVE ********************)
    STATE_JOG_POSITIVE: (* STATE: Start jog movement in positive direction *)
        MC_MoveVelocity_0.Velocity      := Axis[AXIS_INDEX].Parameter.JogVelocity;
        MC_MoveVelocity_0.Acceleration  := Axis[AXIS_INDEX].Parameter.Acceleration;
        MC_MoveVelocity_0.Deceleration  := Axis[AXIS_INDEX].Parameter.Deceleration;
        MC_MoveVelocity_0.Direction     := mcPOSITIVE_DIR;
        MC_MoveVelocity_0.Execute := 1;

        (* check if jog movement should be stopped *)
        IF (Axis[AXIS_INDEX].Command.MoveJogPos = FALSE) THEN
            MC_MoveVelocity_0.Execute := FALSE;
            AxisStep := STATE_HALT;
        END_IF

        IF ((MC_MoveVelocity_0.Error = TRUE) OR (MC_MoveVelocity_0.CommandAborted = TRUE)) THEN
            MC_MoveVelocity_0.Execute := FALSE;
            AxisStep := STATE_READY;
        END_IF

        (* End of STATE_JOG_POSITIVE *)

(********************START JOG MOVEMENT NEGATIVE ********************)
    STATE_JOG_NEGATIVE: (* STATE: Start jog movement in negative direction *)
        MC_MoveVelocity_0.Velocity      := Axis[AXIS_INDEX].Parameter.JogVelocity;
        MC_MoveVelocity_0.Acceleration  := Axis[AXIS_INDEX].Parameter.Acceleration;
        MC_MoveVelocity_0.Deceleration  := Axis[AXIS_INDEX].Parameter.Deceleration;
        MC_MoveVelocity_0.Direction     := mcNEGATIVE_DIR;
        MC_MoveVelocity_0.Execute := 1;

        (* check if jog movement should be stopped *)
        IF (Axis[AXIS_INDEX].Command.MoveJogNeg = FALSE) THEN
            MC_MoveVelocity_0.Execute := FALSE;
            AxisStep := STATE_HALT;
        END_IF

        IF ((MC_MoveVelocity_0.Error = TRUE) OR (MC_MoveVelocity_0.CommandAborted = TRUE)) THEN
            MC_MoveVelocity_0.Execute := FALSE;
            AxisStep := STATE_READY;
        END_IF

        (* End of STATE_JOG_NEGATIVE *)

(********************* START ABSOLUTE MOVEMENT **********************)
    STATE_MOVE_ABSOLUTE: (* STATE: Start absolute movement *)
        MC_MoveAbsolute_0.Position      := Axis[AXIS_INDEX].Parameter.Position;
        MC_MoveAbsolute_0.Velocity      := Axis[AXIS_INDEX].Parameter.Velocity;
        MC_MoveAbsolute_0.Acceleration  := Axis[AXIS_INDEX].Parameter.Acceleration;
        MC_MoveAbsolute_0.Deceleration  := Axis[AXIS_INDEX].Parameter.Deceleration;
        MC_MoveAbsolute_0.Direction     := Axis[AXIS_INDEX].Parameter.Direction;
        MC_MoveAbsolute_0.Execute := 1;

        IF (Axis[AXIS_INDEX].Command.Halt = TRUE) THEN
            Axis[AXIS_INDEX].Command.Halt := 0;
            MC_MoveAbsolute_0.Execute := 0;
            AxisStep := STATE_HALT;
        ELSIF (MC_MoveAbsolute_0.Done = TRUE) THEN
            MC_MoveAbsolute_0.Execute := FALSE;
            AxisStep := STATE_READY;
        END_IF

        IF ((MC_MoveAbsolute_0.Error = TRUE) OR (MC_MoveAbsolute_0.CommandAborted = TRUE)) THEN
            MC_MoveAbsolute_0.Execute := FALSE;
            AxisStep := STATE_READY;
        END_IF

        (* End of STATE_MOVE_ABSOLUTE *)

(********************* START ADDITIVE MOVEMENT **********************)
    STATE_MOVE_ADDITIVE: (* STATE: Start additive movement *)
        MC_MoveAdditive_0.Distance      := Axis[AXIS_INDEX].Parameter.Distance;
        MC_MoveAdditive_0.Velocity      := Axis[AXIS_INDEX].Parameter.Velocity;
        MC_MoveAdditive_0.Acceleration  := Axis[AXIS_INDEX].Parameter.Acceleration;
        MC_MoveAdditive_0.Deceleration  := Axis[AXIS_INDEX].Parameter.Deceleration;
        MC_MoveAdditive_0.Execute := 1;
        IF (Axis[AXIS_INDEX].Command.Halt = TRUE) THEN
            Axis[AXIS_INDEX].Command.Halt := FALSE;
            MC_MoveAdditive_0.Execute := FALSE;
            AxisStep := STATE_HALT;
        ELSIF (MC_MoveAdditive_0.Done = TRUE) THEN
            MC_MoveAdditive_0.Execute := FALSE;
             AxisStep := STATE_READY;
        END_IF

        (* check IF error occured *)
        IF ((MC_MoveAdditive_0.Error = TRUE) OR (MC_MoveAdditive_0.CommandAborted = TRUE)) THEN
            MC_MoveAdditive_0.Execute := FALSE;
            AxisStep := STATE_READY;
        END_IF

        (* End of STATE_MOVE_ADDITIVE *)

(********************* START VELOCITY MOVEMENT **********************)
    STATE_MOVE_VELOCITY: (* STATE: Start velocity movement *)
        MC_MoveVelocity_0.Velocity      := Axis[AXIS_INDEX].Parameter.Velocity;
        MC_MoveVelocity_0.Acceleration  := Axis[AXIS_INDEX].Parameter.Acceleration;
        MC_MoveVelocity_0.Deceleration  := Axis[AXIS_INDEX].Parameter.Deceleration;
        MC_MoveVelocity_0.Direction     := Axis[AXIS_INDEX].Parameter.Direction;
        MC_MoveVelocity_0.Execute := 1;

        IF (Axis[AXIS_INDEX].Command.Halt = TRUE) THEN
            Axis[AXIS_INDEX].Command.Halt := FALSE;
            MC_MoveVelocity_0.Execute := FALSE;
            AxisStep := STATE_HALT;
        ELSIF (MC_MoveVelocity_0.InVelocity = TRUE) THEN
            MC_MoveVelocity_0.Execute := FALSE;
             AxisStep := STATE_READY;
        END_IF
        (* check if error occured *)
        IF ((MC_MoveVelocity_0.Error = TRUE) OR (MC_MoveVelocity_0.CommandAborted = TRUE)) THEN
            MC_MoveVelocity_0.Execute := FALSE;
            AxisStep := STATE_READY;
        END_IF

        (* End of STATE_MOVE_ADDITIVE *)

(*********************** SEQUENCE END *******************************)
END_CASE

(*********************************************************************
        Function Block Calls
*********************************************************************)

(*************************** MC_POWER *******************************)
MC_Power_0.Axis := AxisRef[AXIS_INDEX];
MC_Power_0();

(**************************** MC_HOME *******************************)
MC_Home_0.Axis := AxisRef[AXIS_INDEX];
MC_Home_0();

(************************ MC_MOVEABSOLUTE ***************************)
MC_MoveAbsolute_0.Axis := AxisRef[AXIS_INDEX];
MC_MoveAbsolute_0();

(************************ MC_MOVEADDITIVE ***************************)
MC_MoveAdditive_0.Axis := AxisRef[AXIS_INDEX];
MC_MoveAdditive_0();

(************************ MC_MOVEVELOCITY ***************************)
MC_MoveVelocity_0.Axis := AxisRef[AXIS_INDEX];
MC_MoveVelocity_0();

(**************************** MC_STOP *******************************)
MC_Stop_0.Axis := AxisRef[AXIS_INDEX];
MC_Stop_0();

(****************************MC_HALT*********************************)
MC_Halt_0.Axis := AxisRef[AXIS_INDEX];
MC_Halt_0();

END_PROGRAM
```

#### axisInit.st
```iecst
(********************************************************************
 * COPYRIGHT -- Bernecker + Rainer
 ********************************************************************
 * Program: Axis_01
 * File: axisInit.st
 * Author: Bernecker + Rainer
 * Created: March 01, 2011
 ********************************************************************
 * Implementation of program Axis_01
 ********************************************************************)

PROGRAM _INIT
AxisStep := STATE_WAIT; (* start step *)

Axis[AXIS_INDEX].Parameter.Velocity       := 1000; (* velocity for movement *)
Axis[AXIS_INDEX].Parameter.Acceleration   := 5000; (* acceleration for movement *)
Axis[AXIS_INDEX].Parameter.Deceleration   := 5000; (* deceleration for movement *)
Axis[AXIS_INDEX].Parameter.JogVelocity    := 400;  (* velocity for jogging *)
END_PROGRAM
```

### Program Logical/LibACP10MC_MotionControl_ST/Master_00 (IEC) - master axis handle

#### masterCyclic.st - Cyclic code
```iecst
(********************************************************************
 * COPYRIGHT -- Bernecker + Rainer
 ********************************************************************
 * Program: Master_00
 * File: masterCyclic.st
 * Author: Bernecker + Rainer
 * Created: March 01, 2011
 ********************************************************************
 * Implementation of program Master_00
 ********************************************************************)

PROGRAM _CYCLIC

(************CHECK IF POWER SHOULD BE OFF ***************************)
    IF ((GlobalCommand.Power = FALSE) AND (Master[MASTER_INDEX].Command.Power = FALSE)) THEN
        MasterStep := STATE_WAIT;
    END_IF

    (* central monitoring of the stop command allows a shorter reaction time *)
    IF ((GlobalCommand.Stop = TRUE) OR (Master[MASTER_INDEX].Command.Stop = TRUE)) THEN
        IF ((GlobalCommand.Power = TRUE) OR (Master[MASTER_INDEX].Command.Power = TRUE)) THEN
            MasterStep := STATE_STOP;
            (* reset all FB execute inputs we use *)
            MC_Home_0.Execute := FALSE;
            MC_Halt_0.Execute := FALSE;
            MC_MoveAbsolute_0.Execute := FALSE;
            MC_MoveAdditive_0.Execute := FALSE;
            MC_MoveVelocity_0.Execute := FALSE;

            Master[MASTER_INDEX].Command.MoveJogPos := FALSE;
            Master[MASTER_INDEX].Command.MoveJogNeg := FALSE;
        END_IF
    END_IF

(************************** MC_READSTATUS ***************************)
MC_ReadStatus_0.Enable := NOT(MC_ReadStatus_0.Error);
MC_ReadStatus_0.Axis := MasterRef[MASTER_INDEX];
MC_ReadStatus_0();
Master[MASTER_INDEX].AxisState.Disabled             := MC_ReadStatus_0.Disabled;
Master[MASTER_INDEX].AxisState.StandStill           := MC_ReadStatus_0.StandStill;
Master[MASTER_INDEX].AxisState.Stopping             := MC_ReadStatus_0.Stopping;
Master[MASTER_INDEX].AxisState.Homing               := MC_ReadStatus_0.Homing;
Master[MASTER_INDEX].AxisState.DiscreteMotion       := MC_ReadStatus_0.DiscreteMotion;
Master[MASTER_INDEX].AxisState.ContinuousMotion     := MC_ReadStatus_0.ContinuousMotion;
Master[MASTER_INDEX].AxisState.SynchronizedMotion   := MC_ReadStatus_0.SynchronizedMotion;
Master[MASTER_INDEX].AxisState.ErrorStop            := MC_ReadStatus_0.Errorstop;

(********************** MC_BR_READDRIVESTATUS ***********************)
MC_BR_ReadDriveStatus_0.Enable := NOT(MC_BR_ReadDriveStatus_0.Error);
MC_BR_ReadDriveStatus_0.Axis := MasterRef[MASTER_INDEX];
MC_BR_ReadDriveStatus_0.AdrDriveStatus := ADR(Master[MASTER_INDEX].Status.DriveStatus);
MC_BR_ReadDriveStatus_0();

(********************* MC_READACTUALPOSITION ************************)
MC_ReadActualPosition_0.Enable := NOT(MC_ReadActualPosition_0.Error);
MC_ReadActualPosition_0.Axis := MasterRef[MASTER_INDEX];
MC_ReadActualPosition_0();
IF(MC_ReadActualPosition_0.Valid = TRUE) THEN
    Master[MASTER_INDEX].Status.ActPosition := MC_ReadActualPosition_0.Position;
END_IF

(********************* MC_READACTUALVELOCITY ************************)
MC_ReadActualVelocity_0.Enable := NOT(MC_ReadActualVelocity_0.Error);
MC_ReadActualVelocity_0.Axis := MasterRef[MASTER_INDEX];
MC_ReadActualVelocity_0();
IF(MC_ReadActualVelocity_0.Valid = TRUE) THEN
    Master[MASTER_INDEX].Status.ActVelocity := MC_ReadActualVelocity_0.Velocity;
END_IF

CASE MasterStep OF
(****************************** WAIT ********************************)
    STATE_WAIT: (* STATE: Wait *)
        IF ((GlobalCommand.Power = TRUE) OR (Master[MASTER_INDEX].Command.Power = TRUE)) THEN
            MasterStep := STATE_POWER_ON;
        ELSE
            MC_Power_0.Enable := FALSE;
        END_IF

        (* reset all FB execute inputs we use *)
        MC_Home_0.Execute := FALSE;
        MC_Halt_0.Execute := FALSE;
        MC_Stop_0.Execute := FALSE;
        MC_MoveAbsolute_0.Execute := FALSE;
        MC_MoveAdditive_0.Execute := FALSE;
        MC_MoveVelocity_0.Execute := FALSE;

        (* reset user commands *)
        Master[MASTER_INDEX].Command.Stop := FALSE;
        Master[MASTER_INDEX].Command.MoveJogPos := FALSE;
        Master[MASTER_INDEX].Command.MoveJogNeg := FALSE;
        Master[MASTER_INDEX].Command.MoveVelocity := FALSE;
        Master[MASTER_INDEX].Command.MoveAbsolute := FALSE;
        Master[MASTER_INDEX].Command.MoveAdditive := FALSE;

    (* End of STATE_WAIT *)

(****************************** POWER ON ****************************)
    STATE_POWER_ON: (* STATE: Power on *)
        IF (PowerSupplyOn = TRUE) THEN
            MC_Power_0.Enable := TRUE;
        END_IF
        IF (MC_Power_0.Status = TRUE) THEN
            MasterStep := STATE_READY;
        END_IF

        (* if a power error occured switch off controller *)
        IF (MC_Power_0.Error = TRUE) THEN
            MC_Power_0.Enable := FALSE;
        END_IF

        (* End of STATE_POWER_ON *)

(****************************** READY *******************************)
    STATE_READY: (* STATE: Waiting for Commands *)
        IF ((Master[MASTER_INDEX].Command.Home = TRUE) OR (GlobalCommand.Home = TRUE)) THEN
            Master[MASTER_INDEX].Command.Home := FALSE;
            MasterStep := STATE_HOME;
        ELSIF ((Master[MASTER_INDEX].Command.Stop = TRUE) OR (GlobalCommand.Stop = TRUE)) THEN
            MasterStep := STATE_STOP;
        ELSIF (Master[MASTER_INDEX].Command.MoveJogPos = TRUE) THEN
            MasterStep := STATE_JOG_POSITIVE;
        ELSIF (Master[MASTER_INDEX].Command.MoveJogNeg = TRUE) THEN
            MasterStep := STATE_JOG_NEGATIVE;
        ELSIF (Master[MASTER_INDEX].Command.MoveAbsolute = TRUE) THEN
            Master[MASTER_INDEX].Command.MoveAbsolute := FALSE;
            MasterStep := STATE_MOVE_ABSOLUTE;
        ELSIF (Master[MASTER_INDEX].Command.MoveAdditive = TRUE) THEN
            Master[MASTER_INDEX].Command.MoveAdditive := FALSE;
            MasterStep := STATE_MOVE_ADDITIVE;
        ELSIF (Master[MASTER_INDEX].Command.MoveVelocity = TRUE) THEN
            Master[MASTER_INDEX].Command.MoveVelocity := FALSE;
            MasterStep := STATE_MOVE_VELOCITY;
        ELSIF (Master[MASTER_INDEX].Command.Halt = TRUE) THEN
            Master[MASTER_INDEX].Command.Halt := FALSE;
            MasterStep := STATE_HALT;
        END_IF

        (* End of STATE_READY *)

(****************************** HOME ********************************)
    STATE_HOME: (* STATE: start homing process *)
        MC_Home_0.Position := Master[MASTER_INDEX].Parameter.HomePosition;
        MC_Home_0.HomingMode := Master[MASTER_INDEX].Parameter.HomeMode;
        MC_Home_0.Execute := TRUE;
        IF (MC_Home_0.Done = TRUE) THEN
            GlobalCommand.Home := FALSE;
            MC_Home_0.Execute := FALSE;
            MasterStep := STATE_READY;
        END_IF

        (* if a homing error occured go to ready state *)
        IF ((MC_Home_0.Error = TRUE) OR (MC_Home_0.CommandAborted = TRUE)) THEN
            MC_Home_0.Execute := FALSE;
            MasterStep := STATE_READY;
        END_IF

        (* End of STATE_HOME *)

(*************************** HALT MOVEMENT **************************)
    STATE_HALT: (* STATE: Stop the active movement *)
        MC_Halt_0.Deceleration := Master[MASTER_INDEX].Parameter.Deceleration;
        MC_Halt_0.Execute := TRUE;
        IF (MC_Halt_0.Done = TRUE) THEN
            MC_Halt_0.Execute := FALSE;
            MasterStep := STATE_READY;
       END_IF

       (* check if error occured *)
       IF ((MC_Halt_0.Error = TRUE) OR (MC_Halt_0.CommandAborted = TRUE)) THEN
           MC_Halt_0.Execute := FALSE;
           MasterStep := STATE_READY;
       END_IF

       (* End of STATE_HALT *)

(*************************** STOP MOVEMENT **************************)
    STATE_STOP: (* STATE: Stop movement as long as command is set *)
        MC_Stop_0.Deceleration := Master[MASTER_INDEX].Parameter.Deceleration;
        MC_Stop_0.Execute := TRUE;

        (* if axis is stopped go to ready state *)
        IF ((MC_Stop_0.Done = TRUE) AND (Master[MASTER_INDEX].Command.Stop = FALSE) AND (GlobalCommand.Stop = FALSE)) THEN
            MC_Stop_0.Execute := FALSE;
            MasterStep := STATE_READY;
        END_IF

        (* check if error occured *)
        IF (((MC_Stop_0.Error = TRUE) OR (MC_Stop_0.CommandAborted = TRUE)) AND
             (Master[MASTER_INDEX].Command.Stop = FALSE) AND
             (GlobalCommand.Stop = FALSE)) THEN
            MC_Stop_0.Execute := FALSE;
            MasterStep := STATE_READY;
        END_IF

       (* End of STATE_STOP *)

(******************* START JOG MOVEMENT POSITIVE ********************)
    STATE_JOG_POSITIVE: (* STATE: Start jog movement in positive direction *)
        MC_MoveVelocity_0.Velocity      := Master[MASTER_INDEX].Parameter.JogVelocity;
        MC_MoveVelocity_0.Acceleration  := Master[MASTER_INDEX].Parameter.Acceleration;
        MC_MoveVelocity_0.Deceleration  := Master[MASTER_INDEX].Parameter.Deceleration;
        MC_MoveVelocity_0.Direction     := mcPOSITIVE_DIR;
        MC_MoveVelocity_0.Execute := 1;

        (* check if jog movement should be stopped *)
        IF (Master[MASTER_INDEX].Command.MoveJogPos = FALSE) THEN
            MC_MoveVelocity_0.Execute := FALSE;
            MasterStep := STATE_HALT;
        END_IF

        IF ((MC_MoveVelocity_0.Error = TRUE) OR (MC_MoveVelocity_0.CommandAborted = TRUE)) THEN
            MC_MoveVelocity_0.Execute := FALSE;
            MasterStep := STATE_READY;
        END_IF

        (* End of STATE_JOG_POSITIVE *)

(********************START JOG MOVEMENT NEGATIVE ********************)
    STATE_JOG_NEGATIVE: (* STATE: Start jog movement in negative direction *)
        MC_MoveVelocity_0.Velocity      := Master[MASTER_INDEX].Parameter.JogVelocity;
        MC_MoveVelocity_0.Acceleration  := Master[MASTER_INDEX].Parameter.Acceleration;
        MC_MoveVelocity_0.Deceleration  := Master[MASTER_INDEX].Parameter.Deceleration;
        MC_MoveVelocity_0.Direction     := mcNEGATIVE_DIR;
        MC_MoveVelocity_0.Execute := 1;

        (* check if jog movement should be stopped *)
        IF (Master[MASTER_INDEX].Command.MoveJogNeg = FALSE) THEN
            MC_MoveVelocity_0.Execute := FALSE;
            MasterStep := STATE_HALT;
        END_IF

        IF ((MC_MoveVelocity_0.Error = TRUE) OR (MC_MoveVelocity_0.CommandAborted = TRUE)) THEN
            MC_MoveVelocity_0.Execute := FALSE;
            MasterStep := STATE_READY;
        END_IF

        (* End of STATE_JOG_NEGATIVE *)

(********************* START ABSOLUTE MOVEMENT **********************)
    STATE_MOVE_ABSOLUTE: (* STATE: Start absolute movement *)
        MC_MoveAbsolute_0.Position      := Master[MASTER_INDEX].Parameter.Position;
        MC_MoveAbsolute_0.Velocity      := Master[MASTER_INDEX].Parameter.Velocity;
        MC_MoveAbsolute_0.Acceleration  := Master[MASTER_INDEX].Parameter.Acceleration;
        MC_MoveAbsolute_0.Deceleration  := Master[MASTER_INDEX].Parameter.Deceleration;
        MC_MoveAbsolute_0.Direction     := Master[MASTER_INDEX].Parameter.Direction;
        MC_MoveAbsolute_0.Execute := 1;

        IF (Master[MASTER_INDEX].Command.Halt = TRUE) THEN
            Master[MASTER_INDEX].Command.Halt := 0;
            MC_MoveAbsolute_0.Execute := 0;
            MasterStep := STATE_HALT;
        ELSIF (MC_MoveAbsolute_0.Done = TRUE) THEN
            MC_MoveAbsolute_0.Execute := FALSE;
            MasterStep := STATE_READY;
        END_IF

        IF ((MC_MoveAbsolute_0.Error = TRUE) OR (MC_MoveAbsolute_0.CommandAborted = TRUE)) THEN
            MC_MoveAbsolute_0.Execute := FALSE;
            MasterStep := STATE_READY;
        END_IF

        (* End of STATE_MOVE_ABSOLUTE *)

(********************* START ADDITIVE MOVEMENT **********************)
    STATE_MOVE_ADDITIVE: (* STATE: Start additive movement *)
        MC_MoveAdditive_0.Distance      := Master[MASTER_INDEX].Parameter.Distance;
        MC_MoveAdditive_0.Velocity      := Master[MASTER_INDEX].Parameter.Velocity;
        MC_MoveAdditive_0.Acceleration  := Master[MASTER_INDEX].Parameter.Acceleration;
        MC_MoveAdditive_0.Deceleration  := Master[MASTER_INDEX].Parameter.Deceleration;
        MC_MoveAdditive_0.Execute := 1;
        IF (Master[MASTER_INDEX].Command.Halt = TRUE) THEN
            Master[MASTER_INDEX].Command.Halt := FALSE;
            MC_MoveAdditive_0.Execute := FALSE;
            MasterStep := STATE_HALT;
        ELSIF (MC_MoveAdditive_0.Done = TRUE) THEN
            MC_MoveAdditive_0.Execute := FALSE;
             MasterStep := STATE_READY;
        END_IF

        (* check IF error occured *)
        IF ((MC_MoveAdditive_0.Error = TRUE) OR (MC_MoveAdditive_0.CommandAborted = TRUE)) THEN
            MC_MoveAdditive_0.Execute := FALSE;
            MasterStep := STATE_READY;
        END_IF

        (* End of STATE_MOVE_ADDITIVE *)

(********************* START VELOCITY MOVEMENT **********************)
    STATE_MOVE_VELOCITY: (* STATE: Start velocity movement *)
        MC_MoveVelocity_0.Velocity      := Master[MASTER_INDEX].Parameter.Velocity;
        MC_MoveVelocity_0.Acceleration  := Master[MASTER_INDEX].Parameter.Acceleration;
        MC_MoveVelocity_0.Deceleration  := Master[MASTER_INDEX].Parameter.Deceleration;
        MC_MoveVelocity_0.Direction     := Master[MASTER_INDEX].Parameter.Direction;
        MC_MoveVelocity_0.Execute := 1;

        IF (Master[MASTER_INDEX].Command.Halt = TRUE) THEN
            Master[MASTER_INDEX].Command.Halt := FALSE;
            MC_MoveVelocity_0.Execute := FALSE;
            MasterStep := STATE_HALT;
        ELSIF (MC_MoveVelocity_0.InVelocity = TRUE) THEN
            MC_MoveVelocity_0.Execute := FALSE;
             MasterStep := STATE_READY;
        END_IF
        (* check if error occured *)
        IF ((MC_MoveVelocity_0.Error = TRUE) OR (MC_MoveVelocity_0.CommandAborted = TRUE)) THEN
            MC_MoveVelocity_0.Execute := FALSE;
            MasterStep := STATE_READY;
        END_IF

        (* End of STATE_MOVE_ADDITIVE *)

(*********************** SEQUENCE END *******************************)
END_CASE

(*********************************************************************
        Function Block Calls
*********************************************************************)

(*************************** MC_POWER *******************************)
MC_Power_0.Axis := MasterRef[MASTER_INDEX];
MC_Power_0();

(**************************** MC_HOME *******************************)
MC_Home_0.Axis := MasterRef[MASTER_INDEX];
MC_Home_0();

(************************ MC_MOVEABSOLUTE ***************************)
MC_MoveAbsolute_0.Axis := MasterRef[MASTER_INDEX];
MC_MoveAbsolute_0();

(************************ MC_MOVEADDITIVE ***************************)
MC_MoveAdditive_0.Axis := MasterRef[MASTER_INDEX];
MC_MoveAdditive_0();

(************************ MC_MOVEVELOCITY ***************************)
MC_MoveVelocity_0.Axis := MasterRef[MASTER_INDEX];
MC_MoveVelocity_0();

(**************************** MC_STOP *******************************)
MC_Stop_0.Axis := MasterRef[MASTER_INDEX];
MC_Stop_0();

(*************************** MC_HALT ********************************)
MC_Halt_0.Axis := MasterRef[MASTER_INDEX];
MC_Halt_0();

END_PROGRAM
```

#### masterInit.st - Initialization code
```iecst
(********************************************************************
 * COPYRIGHT -- Bernecker + Rainer
 ********************************************************************
 * Program: Master_00
 * File: masterInit.st
 * Author: Bernecker + Rainer
 * Created: March 01, 2011
 ********************************************************************
 * Implementation of program Master_00
 ********************************************************************)

PROGRAM _INIT
MasterStep := STATE_WAIT; (* start step *)

Master[MASTER_INDEX].Parameter.Velocity       := 1000; (* velocity for movement *)
Master[MASTER_INDEX].Parameter.Acceleration   := 5000; (* acceleration for movement *)
Master[MASTER_INDEX].Parameter.Deceleration   := 5000; (* deceleration for movement *)
Master[MASTER_INDEX].Parameter.JogVelocity    := 400;  (* velocity for jogging *)
END_PROGRAM
```

#### master.var - Local variables
```iecst
(*Actual step inside the step sequencer*)
VAR
	MasterStep : USINT; (*current step in the step sequence*)
END_VAR
VAR CONSTANT
	STATE_WAIT : USINT := 0; (*constant for a waiting step*)
	STATE_POWER_ON : USINT := 1; (*constant for the step in which the controller is switched on*)
	STATE_HOME : USINT := 2; (*constant for the step in which the axis is referenced*)
	STATE_READY : USINT := 10; (*constant for a waiting step*)
	STATE_HALT : USINT := 11; (*constant for the step in which movements are stopped*)
	STATE_STOP : USINT := 12; (*constant for the step in which movements are stopped *)
	STATE_JOG_POSITIVE : USINT := 13; (*constant for the step in which positive jogging movement is executed*)
	STATE_JOG_NEGATIVE : USINT := 14; (*constant for the step in which negative jogging movement is executed*)
	STATE_MOVE_ABSOLUTE : USINT := 15; (*constant for the step in which a movement to defined position is executed*)
	STATE_MOVE_ADDITIVE : USINT := 16; (*constant for the step in which a movement with defined distance is executed*)
	STATE_MOVE_VELOCITY : USINT := 17; (*constant for the step in which a movement with defined velocity is started*)
END_VAR
(*Index of the used axis*)
VAR CONSTANT
	MASTER_INDEX : USINT := 0; (*Index of the used axis*)
END_VAR
(*Function Blocks*)
VAR
	MC_BR_ReadDriveStatus_0 : MC_BR_ReadDriveStatus; (*Function Block*)
	MC_Halt_0 : MC_Halt; (*Function Block*)
	MC_Home_0 : MC_Home; (*Function Block*)
	MC_MoveAbsolute_0 : MC_MoveAbsolute; (*Function Block*)
	MC_MoveAdditive_0 : MC_MoveAdditive; (*Function Block*)
	MC_MoveVelocity_0 : MC_MoveVelocity; (*Function Block*)
	MC_Power_0 : MC_Power; (*Function Block*)
	MC_ReadActualPosition_0 : MC_ReadActualPosition; (*Function Block*)
	MC_ReadActualVelocity_0 : MC_ReadActualVelocity; (*Function Block*)
	MC_ReadStatus_0 : MC_ReadStatus; (*Function Block*)
	MC_Stop_0 : MC_Stop; (*Function Block*)
END_VAR
```

### Program Logical/LibACP10MC_MotionControl_ST/Slave_00 (IEC) - slave axis handle

#### slaveCyclic.st - Cyclic code
```iecst
(********************************************************************
 * COPYRIGHT -- Bernecker + Rainer
 ********************************************************************
 * Program: Slave_00
 * File: slaveCyclic.st
 * Author: Bernecker + Rainer
 * Created: March 01, 2011
 ********************************************************************
 * Implementation of program Slave_00
 ********************************************************************)

PROGRAM _CYCLIC

(************CHECK IF POWER SHOULD BE OFF ***************************)
    IF ((GlobalCommand.Power = FALSE) AND (Slave[SLAVE_INDEX].Command.Power = FALSE)) THEN
        SlaveStep := STATE_WAIT;
    END_IF

    (* central monitoring of the stop command allows a shorter reaction time *)
    IF ((GlobalCommand.Stop = TRUE) OR (Slave[SLAVE_INDEX].Command.Stop = TRUE)) THEN
        IF ((GlobalCommand.Power = TRUE) OR (Slave[SLAVE_INDEX].Command.Power = TRUE)) THEN
            SlaveStep := STATE_STOP;
            (* reset all FB execute inputs we use *)
            MC_Home_0.Execute := FALSE;
            MC_Halt_0.Execute := FALSE;
            MC_MoveAbsolute_0.Execute := FALSE;
            MC_MoveAdditive_0.Execute := FALSE;
            MC_MoveVelocity_0.Execute := FALSE;

            MC_BR_InitAutData_0.Execute := FALSE;
            MC_BR_AutCommand_0.Enable := FALSE;
            MC_BR_AutCommand_0.Start := FALSE;
            MC_BR_AutCommand_0.Restart := FALSE;
            MC_BR_AutCommand_0.Stop := FALSE;
            MC_BR_AutCommand_0.EndAutomat := FALSE;

            Slave[SLAVE_INDEX].Command.MoveJogPos := FALSE;
            Slave[SLAVE_INDEX].Command.MoveJogNeg := FALSE;
        END_IF
    END_IF

(************************** MC_READSTATUS ***************************)
MC_ReadStatus_0.Enable := NOT(MC_ReadStatus_0.Error);
MC_ReadStatus_0.Axis := SlaveRef[SLAVE_INDEX];
MC_ReadStatus_0();
Slave[SLAVE_INDEX].AxisState.Disabled             := MC_ReadStatus_0.Disabled;
Slave[SLAVE_INDEX].AxisState.StandStill           := MC_ReadStatus_0.StandStill;
Slave[SLAVE_INDEX].AxisState.Stopping             := MC_ReadStatus_0.Stopping;
Slave[SLAVE_INDEX].AxisState.Homing               := MC_ReadStatus_0.Homing;
Slave[SLAVE_INDEX].AxisState.DiscreteMotion       := MC_ReadStatus_0.DiscreteMotion;
Slave[SLAVE_INDEX].AxisState.ContinuousMotion     := MC_ReadStatus_0.ContinuousMotion;
Slave[SLAVE_INDEX].AxisState.SynchronizedMotion   := MC_ReadStatus_0.SynchronizedMotion;
Slave[SLAVE_INDEX].AxisState.ErrorStop            := MC_ReadStatus_0.Errorstop;

(********************** MC_BR_READDRIVESTATUS ***********************)
MC_BR_ReadDriveStatus_0.Enable := NOT(MC_BR_ReadDriveStatus_0.Error);
MC_BR_ReadDriveStatus_0.Axis := SlaveRef[SLAVE_INDEX];
MC_BR_ReadDriveStatus_0.AdrDriveStatus := ADR(Slave[SLAVE_INDEX].Status.DriveStatus);
MC_BR_ReadDriveStatus_0();

(********************* MC_READACTUALPOSITION ************************)
MC_ReadActualPosition_0.Enable := NOT(MC_ReadActualPosition_0.Error);
MC_ReadActualPosition_0.Axis := SlaveRef[SLAVE_INDEX];
MC_ReadActualPosition_0();
IF(MC_ReadActualPosition_0.Valid = TRUE) THEN
    Slave[SLAVE_INDEX].Status.ActPosition := MC_ReadActualPosition_0.Position;
END_IF

(********************* MC_READACTUALVELOCITY ************************)
MC_ReadActualVelocity_0.Enable := NOT(MC_ReadActualVelocity_0.Error);
MC_ReadActualVelocity_0.Axis := SlaveRef[SLAVE_INDEX];
MC_ReadActualVelocity_0();
IF(MC_ReadActualVelocity_0.Valid = TRUE) THEN
    Slave[SLAVE_INDEX].Status.ActVelocity := MC_ReadActualVelocity_0.Velocity;
END_IF

CASE SlaveStep OF
(****************************** WAIT ********************************)
    STATE_WAIT: (* STATE: Wait *)
        IF ((GlobalCommand.Power = TRUE) OR (Slave[SLAVE_INDEX].Command.Power = TRUE)) THEN
            SlaveStep := STATE_POWER_ON;
        ELSE
            MC_Power_0.Enable := FALSE;
        END_IF

        (* reset all FB execute inputs we use *)
        MC_Home_0.Execute := FALSE;
        MC_Halt_0.Execute := FALSE;
        MC_Stop_0.Execute := FALSE;
        MC_MoveAbsolute_0.Execute := FALSE;
        MC_MoveAdditive_0.Execute := FALSE;
        MC_MoveVelocity_0.Execute := FALSE;

        (* reset user commands *)
        Slave[SLAVE_INDEX].Command.Stop := FALSE;
        Slave[SLAVE_INDEX].Command.MoveJogPos := FALSE;
        Slave[SLAVE_INDEX].Command.MoveJogNeg := FALSE;
        Slave[SLAVE_INDEX].Command.MoveVelocity := FALSE;
        Slave[SLAVE_INDEX].Command.MoveAbsolute := FALSE;
        Slave[SLAVE_INDEX].Command.MoveAdditive := FALSE;

    (* End of STATE_WAIT *)

(****************************** POWER ON ****************************)
    STATE_POWER_ON: (* STATE: Power on *)
        IF (PowerSupplyOn = TRUE) THEN
            MC_Power_0.Enable := TRUE;
        END_IF
        IF (MC_Power_0.Status = TRUE) THEN
            SlaveStep := STATE_READY;
        END_IF

        (* if a power error occured switch off controller *)
        IF (MC_Power_0.Error = TRUE) THEN
            MC_Power_0.Enable := FALSE;
        END_IF

        (* End of STATE_POWER_ON *)

(****************************** READY *******************************)
    STATE_READY: (* STATE: Waiting for Commands *)
        IF ((Slave[SLAVE_INDEX].Command.Home = TRUE) OR (GlobalCommand.Home = TRUE)) THEN
            Slave[SLAVE_INDEX].Command.Home := FALSE;
            SlaveStep := STATE_HOME;
        ELSIF ((Slave[SLAVE_INDEX].Command.Stop = TRUE) OR (GlobalCommand.Stop = TRUE)) THEN
            SlaveStep := STATE_STOP;
        ELSIF (Slave[SLAVE_INDEX].Command.MoveJogPos = TRUE) THEN
            SlaveStep := STATE_JOG_POSITIVE;
        ELSIF (Slave[SLAVE_INDEX].Command.MoveJogNeg = TRUE) THEN
            SlaveStep := STATE_JOG_NEGATIVE;
        ELSIF (Slave[SLAVE_INDEX].Command.MoveAbsolute = TRUE) THEN
            Slave[SLAVE_INDEX].Command.MoveAbsolute := FALSE;
            SlaveStep := STATE_MOVE_ABSOLUTE;
        ELSIF (Slave[SLAVE_INDEX].Command.MoveAdditive = TRUE) THEN
            Slave[SLAVE_INDEX].Command.MoveAdditive := FALSE;
            SlaveStep := STATE_MOVE_ADDITIVE;
        ELSIF (Slave[SLAVE_INDEX].Command.MoveVelocity = TRUE) THEN
            Slave[SLAVE_INDEX].Command.MoveVelocity := FALSE;
            SlaveStep := STATE_MOVE_VELOCITY;
        ELSIF (Slave[SLAVE_INDEX].Command.Halt = TRUE) THEN
            Slave[SLAVE_INDEX].Command.Halt := FALSE;
            SlaveStep := STATE_HALT;
        ELSIF (Slave[SLAVE_INDEX].Command.StartAutomat = TRUE) THEN
            Slave[SLAVE_INDEX].Command.StartAutomat := FALSE;
            SlaveStep := STATE_AUTOMAT_INIT;
        ELSIF (Slave[SLAVE_INDEX].Command.RestartAutomat = TRUE) THEN
            Slave[SLAVE_INDEX].Command.RestartAutomat := FALSE;
            SlaveStep := STATE_AUTOMAT_RESTART;
        ELSIF (Slave[SLAVE_INDEX].Command.EndAutomat = TRUE) THEN
            Slave[SLAVE_INDEX].Command.EndAutomat := FALSE;
            SlaveStep := STATE_AUTOMAT_END;
        ELSIF (Slave[SLAVE_INDEX].Command.StopSlave = TRUE) THEN
            Slave[SLAVE_INDEX].Command.StopSlave := FALSE;
            SlaveStep := STATE_AUTOMAT_STOP;
        END_IF

        (* End of STATE_READY *)

(****************************** HOME ********************************)
    STATE_HOME: (* STATE: start homing process *)
        MC_Home_0.Position := Slave[SLAVE_INDEX].Parameter.HomePosition;
        MC_Home_0.HomingMode := Slave[SLAVE_INDEX].Parameter.HomeMode;
        MC_Home_0.Execute := TRUE;
        IF (MC_Home_0.Done = TRUE) THEN
            GlobalCommand.Home := FALSE;
            MC_Home_0.Execute := FALSE;
            SlaveStep := STATE_READY;
        END_IF

        (* if a homing error occured go to ready state *)
        IF ((MC_Home_0.Error = TRUE) OR (MC_Home_0.CommandAborted = TRUE)) THEN
            MC_Home_0.Execute := FALSE;
            SlaveStep := STATE_READY;
        END_IF

        (* End of STATE_HOME *)

(*************************** HALT MOVEMENT **************************)
    STATE_HALT: (* STATE: Stop the active movement *)
        MC_Halt_0.Deceleration := Slave[SLAVE_INDEX].Parameter.Deceleration;
        MC_Halt_0.Execute := TRUE;
        IF (MC_Halt_0.Done = TRUE) THEN
            MC_Halt_0.Execute := FALSE;
            SlaveStep := STATE_READY;
       END_IF

       (* check if error occured *)
       IF ((MC_Halt_0.Error = TRUE) OR (MC_Halt_0.CommandAborted = TRUE)) THEN
           MC_Halt_0.Execute := FALSE;
           SlaveStep := STATE_READY;
       END_IF

       (* End of STATE_HALT *)

(*************************** STOP MOVEMENT **************************)
    STATE_STOP: (* STATE: Stop movement as long as command is set *)
        MC_Stop_0.Deceleration := Slave[SLAVE_INDEX].Parameter.Deceleration;
        MC_Stop_0.Execute := TRUE;

        (* if axis is stopped go to ready state *)
        IF ((MC_Stop_0.Done = TRUE) AND (Slave[SLAVE_INDEX].Command.Stop = FALSE) AND (GlobalCommand.Stop = FALSE)) THEN
            MC_Stop_0.Execute := FALSE;
            SlaveStep := STATE_READY;
        END_IF

        (* check if error occured *)
        IF (((MC_Stop_0.Error = TRUE) OR (MC_Stop_0.CommandAborted = TRUE)) AND
             (Slave[SLAVE_INDEX].Command.Stop = FALSE) AND
             (GlobalCommand.Stop = FALSE)) THEN
            MC_Stop_0.Execute := FALSE;
            SlaveStep := STATE_READY;
        END_IF

       (* End of STATE_STOP *)

(******************* START JOG MOVEMENT POSITIVE ********************)
    STATE_JOG_POSITIVE: (* STATE: Start jog movement in positive direction *)
        MC_MoveVelocity_0.Velocity      := Slave[SLAVE_INDEX].Parameter.JogVelocity;
        MC_MoveVelocity_0.Acceleration  := Slave[SLAVE_INDEX].Parameter.Acceleration;
        MC_MoveVelocity_0.Deceleration  := Slave[SLAVE_INDEX].Parameter.Deceleration;
        MC_MoveVelocity_0.Direction     := mcPOSITIVE_DIR;
        MC_MoveVelocity_0.Execute := 1;

        (* check if jog movement should be stopped *)
        IF (Slave[SLAVE_INDEX].Command.MoveJogPos = FALSE) THEN
            MC_MoveVelocity_0.Execute := FALSE;
            SlaveStep := STATE_HALT;
        END_IF

        IF ((MC_MoveVelocity_0.Error = TRUE) OR (MC_MoveVelocity_0.CommandAborted = TRUE)) THEN
            MC_MoveVelocity_0.Execute := FALSE;
            SlaveStep := STATE_READY;
        END_IF

        (* End of STATE_JOG_POSITIVE *)

(********************START JOG MOVEMENT NEGATIVE ********************)
    STATE_JOG_NEGATIVE: (* STATE: Start jog movement in negative direction *)
        MC_MoveVelocity_0.Velocity      := Slave[SLAVE_INDEX].Parameter.JogVelocity;
        MC_MoveVelocity_0.Acceleration  := Slave[SLAVE_INDEX].Parameter.Acceleration;
        MC_MoveVelocity_0.Deceleration  := Slave[SLAVE_INDEX].Parameter.Deceleration;
        MC_MoveVelocity_0.Direction     := mcNEGATIVE_DIR;
        MC_MoveVelocity_0.Execute := 1;

        (* check if jog movement should be stopped *)
        IF (Slave[SLAVE_INDEX].Command.MoveJogNeg = FALSE) THEN
            MC_MoveVelocity_0.Execute := FALSE;
            SlaveStep := STATE_HALT;
        END_IF

        IF ((MC_MoveVelocity_0.Error = TRUE) OR (MC_MoveVelocity_0.CommandAborted = TRUE)) THEN
            MC_MoveVelocity_0.Execute := FALSE;
            SlaveStep := STATE_READY;
        END_IF

        (* End of STATE_JOG_NEGATIVE *)

(********************* START ABSOLUTE MOVEMENT **********************)
    STATE_MOVE_ABSOLUTE: (* STATE: Start absolute movement *)
        MC_MoveAbsolute_0.Position      := Slave[SLAVE_INDEX].Parameter.Position;
        MC_MoveAbsolute_0.Velocity      := Slave[SLAVE_INDEX].Parameter.Velocity;
        MC_MoveAbsolute_0.Acceleration  := Slave[SLAVE_INDEX].Parameter.Acceleration;
        MC_MoveAbsolute_0.Deceleration  := Slave[SLAVE_INDEX].Parameter.Deceleration;
        MC_MoveAbsolute_0.Direction     := Slave[SLAVE_INDEX].Parameter.Direction;
        MC_MoveAbsolute_0.Execute := 1;

        IF (Slave[SLAVE_INDEX].Command.Halt = TRUE) THEN
            Slave[SLAVE_INDEX].Command.Halt := 0;
            MC_MoveAbsolute_0.Execute := 0;
            SlaveStep := STATE_HALT;
        ELSIF (MC_MoveAbsolute_0.Done = TRUE) THEN
            MC_MoveAbsolute_0.Execute := FALSE;
            SlaveStep := STATE_READY;
        END_IF

        IF ((MC_MoveAbsolute_0.Error = TRUE) OR (MC_MoveAbsolute_0.CommandAborted = TRUE)) THEN
            MC_MoveAbsolute_0.Execute := FALSE;
            SlaveStep := STATE_READY;
        END_IF

        (* End of STATE_MOVE_ABSOLUTE *)

(********************* START ADDITIVE MOVEMENT **********************)
    STATE_MOVE_ADDITIVE: (* STATE: Start additive movement *)
        MC_MoveAdditive_0.Distance      := Slave[SLAVE_INDEX].Parameter.Distance;
        MC_MoveAdditive_0.Velocity      := Slave[SLAVE_INDEX].Parameter.Velocity;
        MC_MoveAdditive_0.Acceleration  := Slave[SLAVE_INDEX].Parameter.Acceleration;
        MC_MoveAdditive_0.Deceleration  := Slave[SLAVE_INDEX].Parameter.Deceleration;
        MC_MoveAdditive_0.Execute := 1;
        IF (Slave[SLAVE_INDEX].Command.Halt = TRUE) THEN
            Slave[SLAVE_INDEX].Command.Halt := FALSE;
            MC_MoveAdditive_0.Execute := FALSE;
            SlaveStep := STATE_HALT;
        ELSIF (MC_MoveAdditive_0.Done = TRUE) THEN
            MC_MoveAdditive_0.Execute := FALSE;
             SlaveStep := STATE_READY;
        END_IF

        (* check IF error occured *)
        IF ((MC_MoveAdditive_0.Error = TRUE) OR (MC_MoveAdditive_0.CommandAborted = TRUE)) THEN
            MC_MoveAdditive_0.Execute := FALSE;
            SlaveStep := STATE_READY;
        END_IF

        (* End of STATE_MOVE_ADDITIVE *)

(********************* START VELOCITY MOVEMENT **********************)
    STATE_MOVE_VELOCITY: (* STATE: Start velocity movement *)
        MC_MoveVelocity_0.Velocity      := Slave[SLAVE_INDEX].Parameter.Velocity;
        MC_MoveVelocity_0.Acceleration  := Slave[SLAVE_INDEX].Parameter.Acceleration;
        MC_MoveVelocity_0.Deceleration  := Slave[SLAVE_INDEX].Parameter.Deceleration;
        MC_MoveVelocity_0.Direction     := Slave[SLAVE_INDEX].Parameter.Direction;
        MC_MoveVelocity_0.Execute := 1;

        IF (Slave[SLAVE_INDEX].Command.Halt = TRUE) THEN
            Slave[SLAVE_INDEX].Command.Halt := FALSE;
            MC_MoveVelocity_0.Execute := FALSE;
            SlaveStep := STATE_HALT;
        ELSIF (MC_MoveVelocity_0.InVelocity = TRUE) THEN
            MC_MoveVelocity_0.Execute := FALSE;
             SlaveStep := STATE_READY;
        END_IF
        (* check if error occured *)
        IF ((MC_MoveVelocity_0.Error = TRUE) OR (MC_MoveVelocity_0.CommandAborted = TRUE)) THEN
            MC_MoveVelocity_0.Execute := FALSE;
            SlaveStep := STATE_READY;
        END_IF

        (* End of STATE_MOVE_ADDITIVE *)

(****************** INITIALIZE AUTOMAT PARAMETERS *******************)
    STATE_AUTOMAT_INIT:
        Labeler(MasterRef[0],AutData); (*Call of the function with the Automat Data*)

        MC_BR_InitAutData_0.InitOptions.GlobalParams      := mcALL_PARAMS;
        MC_BR_InitAutData_0.InitOptions.StateIndex        := mcALL_STATES;
        MC_BR_InitAutData_0.InitOptions.EventIndex        := mcALL_EVENTS;
        MC_BR_InitAutData_0.InitOptions.MaxStatesPerCycle := 14;
        MC_BR_InitAutData_0.InitOptions.Force             := mcOFF;
        MC_BR_InitAutData_0.AdrAutData  := ADR(AutData);
        MC_BR_InitAutData_0.Execute     := TRUE;

        (* wait for initialization done *)
        IF (MC_BR_InitAutData_0.Done = TRUE) THEN
            MC_BR_InitAutData_0.Execute := FALSE;
            SlaveStep := STATE_AUTOMAT_START;
        END_IF

        (* check if error occured *)
        IF (MC_BR_InitAutData_0.Error = TRUE) THEN
            MC_BR_InitAutData_0.Execute := FALSE;
            SlaveStep := STATE_READY;
        END_IF

        (* End of STATE_MOVE_VELOCITY *)

(********************** ENABLE CAM-AUTOMAT **************************)
    STATE_AUTOMAT_START:
        MC_BR_AutCommand_0.Enable := TRUE;
        MC_BR_AutCommand_0.Start := TRUE;

        (* wait for autoamt stop *)
        IF (Slave[SLAVE_INDEX].Command.Halt = TRUE) THEN
            Slave[SLAVE_INDEX].Command.Halt := FALSE;
            MC_BR_AutCommand_0.Enable := FALSE;
            MC_BR_AutCommand_0.Start := FALSE;
            SlaveStep := STATE_HALT;
        ELSIF (MC_BR_AutCommand_0.Running = TRUE) THEN
            MC_BR_AutCommand_0.Start := FALSE;
            SlaveStep := STATE_READY;
        END_IF

        (* check if error occured *)
        IF (MC_BR_AutCommand_0.Error = TRUE) THEN
            MC_BR_AutCommand_0.Enable := FALSE;
            MC_BR_AutCommand_0.Start := FALSE;
            SlaveStep := STATE_READY;
        END_IF

        (* End of STATE_AUTOMAT_START *)

(********************** RESTART CAM-AUTOMAT *************************)
    STATE_AUTOMAT_RESTART:
        IF (MC_BR_AutCommand_0.StandBy = FALSE) THEN
            SlaveStep := STATE_READY;
            RETURN;
        END_IF

        MC_BR_AutCommand_0.Enable := TRUE;
        MC_BR_AutCommand_0.Restart := TRUE;

        (* wait for autoamt stop *)
        IF (Slave[SLAVE_INDEX].Command.Halt = TRUE) THEN
            Slave[SLAVE_INDEX].Command.Halt := FALSE;
            MC_BR_AutCommand_0.Enable := FALSE;
            MC_BR_AutCommand_0.Restart := FALSE;
            SlaveStep := STATE_HALT;
        ELSIF (MC_BR_AutCommand_0.Running = TRUE) THEN
            MC_BR_AutCommand_0.Restart := FALSE;
            SlaveStep := STATE_READY;
        END_IF

        (* check if error occured *)
        IF (MC_BR_AutCommand_0.Error = TRUE) THEN
            MC_BR_AutCommand_0.Enable := FALSE;
            MC_BR_AutCommand_0.Restart := FALSE;
            SlaveStep := STATE_READY;
        END_IF

        (* End of STATE_AUTOMAT_RESTART *)

(*********************** STOP CAM-AUTOMAT ***************************)
    STATE_AUTOMAT_STOP:
        MC_BR_AutCommand_0.Deceleration := Slave[SLAVE_INDEX].Parameter.Deceleration;
        MC_BR_AutCommand_0.Stop := TRUE;

        (* check if automat is stopped *)
        IF (MC_BR_AutCommand_0.Running = FALSE) THEN
            MC_BR_AutCommand_0.Stop := FALSE;
            SlaveStep := STATE_READY;
        END_IF

        IF (MC_BR_AutCommand_0.Error = TRUE) THEN
            MC_BR_AutCommand_0.Enable := FALSE;
            MC_BR_AutCommand_0.Stop := FALSE;
            SlaveStep := STATE_READY;
        END_IF

        (* End of STATE_AUTOMAT_STOP *)

(************************ END CAM-AUTOMAT ***************************)
    STATE_AUTOMAT_END:
        MC_BR_AutCommand_0.Deceleration := Slave[SLAVE_INDEX].Parameter.Deceleration;
        MC_BR_AutCommand_0.Stop := TRUE;

        (* check if automat is stopped *)
        IF (MC_BR_AutCommand_0.Running = FALSE) THEN
            MC_BR_AutCommand_0.Enable := FALSE;
            MC_BR_AutCommand_0.EndAutomat := FALSE;
            SlaveStep := STATE_READY;
        END_IF

        (* check if error occured *)
        IF (MC_BR_AutCommand_0.Error = TRUE) THEN
            MC_BR_AutCommand_0.Enable := FALSE;
            MC_BR_AutCommand_0.EndAutomat := FALSE;
            SlaveStep := STATE_READY;
        END_IF

        (* End of STATE_AUTOMAT_STOP *)

(*********************** SEQUENCE END *******************************)
END_CASE

(*********************************************************************
        Function Block Calls
*********************************************************************)

(*************************** MC_POWER *******************************)
MC_Power_0.Axis := SlaveRef[SLAVE_INDEX];
MC_Power_0();

(**************************** MC_HOME *******************************)
MC_Home_0.Axis := SlaveRef[SLAVE_INDEX];
MC_Home_0();

(************************ MC_MOVEABSOLUTE ***************************)
MC_MoveAbsolute_0.Axis := SlaveRef[SLAVE_INDEX];
MC_MoveAbsolute_0();

(************************ MC_MOVEADDITIVE ***************************)
MC_MoveAdditive_0.Axis := SlaveRef[SLAVE_INDEX];
MC_MoveAdditive_0();

(************************ MC_MOVEVELOCITY ***************************)
MC_MoveVelocity_0.Axis := SlaveRef[SLAVE_INDEX];
MC_MoveVelocity_0();

(**************************** MC_STOP *******************************)
MC_Stop_0.Axis := SlaveRef[SLAVE_INDEX];
MC_Stop_0();

(*************************** MC_HALT ********************************)
MC_Halt_0.Axis := SlaveRef[SLAVE_INDEX];
MC_Halt_0();

(********************** MC_BR_INITAUTDATA ***************************)
MC_BR_InitAutData_0.Slave := SlaveRef[SLAVE_INDEX];
MC_BR_InitAutData_0();

(*********************** MC_BR_AUTCOMMAND ***************************)
MC_BR_AutCommand_0.SetSignal1 := Slave[SLAVE_INDEX].Command.SetSignal1;
MC_BR_AutCommand_0.SetSignal2 := Slave[SLAVE_INDEX].Command.SetSignal2;
MC_BR_AutCommand_0.SetSignal3 := Slave[SLAVE_INDEX].Command.SetSignal3;
MC_BR_AutCommand_0.SetSignal4 := Slave[SLAVE_INDEX].Command.SetSignal4;
MC_BR_AutCommand_0.ResetSignal1 := Slave[SLAVE_INDEX].Command.ResetSignal1;
MC_BR_AutCommand_0.ResetSignal2 := Slave[SLAVE_INDEX].Command.ResetSignal2;
MC_BR_AutCommand_0.ResetSignal3 := Slave[SLAVE_INDEX].Command.ResetSignal3;
MC_BR_AutCommand_0.ResetSignal4 := Slave[SLAVE_INDEX].Command.ResetSignal4;
MC_BR_AutCommand_0.Slave := SlaveRef[SLAVE_INDEX];
MC_BR_AutCommand_0();
Slave[SLAVE_INDEX].Status.AutomatRunning := MC_BR_AutCommand_0.Running;
Slave[SLAVE_INDEX].Status.AutomatStandBy := MC_BR_AutCommand_0.StandBy;
Slave[SLAVE_INDEX].Status.ActualStateIndex := MC_BR_AutCommand_0.ActualStateIndex;
Slave[SLAVE_INDEX].Status.ActualStateCamIndex := MC_BR_AutCommand_0.ActualStateCamIndex;
Slave[SLAVE_INDEX].Status.InCam := MC_BR_AutCommand_0.InCam;
Slave[SLAVE_INDEX].Status.InCompensation := MC_BR_AutCommand_0.InCompensation;
END_PROGRAM
```

#### slaveInit.st - Initialization code
```iecst
(********************************************************************
 * COPYRIGHT -- Bernecker + Rainer
 ********************************************************************
 * Program: Slave_00
 * File: slaveInit.st
 * Author: Bernecker + Rainer
 * Created: March 01, 2011
 ********************************************************************
 * Implementation of program Slave_00
 ********************************************************************)

PROGRAM _INIT
SlaveStep := STATE_WAIT; (* start step *)

Slave[SLAVE_INDEX].Parameter.Velocity       := 1000; (* velocity for movement *)
Slave[SLAVE_INDEX].Parameter.Acceleration   := 5000; (* acceleration for movement *)
Slave[SLAVE_INDEX].Parameter.Deceleration   := 5000; (* deceleration for movement *)
Slave[SLAVE_INDEX].Parameter.JogVelocity    := 400;  (* velocity for jogging *)
END_PROGRAM
```

#### slave.var - Local variables
```iecst
(*Actual step inside step sequencer*)
VAR
	SlaveStep : USINT; (*current  step in the step sequence*)
END_VAR
VAR CONSTANT
	STATE_WAIT : USINT := 0; (*constant for a waiting step*)
	STATE_POWER_ON : USINT := 1; (*constant for the step in which the controller is switched on*)
	STATE_HOME : USINT := 2; (*constant for the step in which the axis is referenced*)
	STATE_READY : USINT := 10; (*constant for a waiting step*)
	STATE_HALT : USINT := 11; (*constant for the step in which movements are stopped*)
	STATE_STOP : USINT := 12; (*constant for the step in which movements are stopped*)
	STATE_JOG_POSITIVE : USINT := 13; (*constant for the step in which positive jogging movement is executed*)
	STATE_JOG_NEGATIVE : USINT := 14; (*constant for the step in which negative jogging movement is executed*)
	STATE_MOVE_ABSOLUTE : USINT := 15; (*constant for the step in which a movement to defined position is executed*)
	STATE_MOVE_ADDITIVE : USINT := 16; (*constant for the step in which a movement with defined distance is executed*)
	STATE_MOVE_VELOCITY : USINT := 17; (*constant for the step in which a movement with defined velocity is started*)
	STATE_AUTOMAT_INIT : USINT := 30; (*constant for the step in which the automat is configured*)
	STATE_AUTOMAT_START : USINT := 31; (*constant for the step in which the automat is started*)
	STATE_AUTOMAT_STOP : USINT := 32; (*constant for the step in which the automat is stopped*)
	STATE_AUTOMAT_RESTART : USINT := 33; (*constant for the step in which the automat is restarted*)
	STATE_AUTOMAT_END : USINT := 34; (*constant for the step in which the automat is finished*)
END_VAR
(*Index of the used axis*)
VAR CONSTANT
	SLAVE_INDEX : USINT := 0; (*Index of the used axis*)
END_VAR
(*Configuration data of the automat*)
VAR
	AutData : MC_AUTDATA_TYP; (*configuration of the automat*)
END_VAR
(*Function Blocks*)
VAR
	MC_BR_AutCommand_0 : MC_BR_AutCommand; (*Function Block*)
	MC_BR_InitAutData_0 : MC_BR_InitAutData; (*Function Block*)
	MC_BR_ReadDriveStatus_0 : MC_BR_ReadDriveStatus; (*Function Block *)
	MC_Halt_0 : MC_Halt; (*Function Block *)
	MC_Home_0 : MC_Home; (*Function Block *)
	MC_MoveAbsolute_0 : MC_MoveAbsolute; (*Function Block *)
	MC_MoveAdditive_0 : MC_MoveAdditive; (*Function Block *)
	MC_MoveVelocity_0 : MC_MoveVelocity; (*Function Block *)
	MC_Power_0 : MC_Power; (*Function Block *)
	MC_ReadActualPosition_0 : MC_ReadActualPosition; (*Function Block *)
	MC_ReadActualVelocity_0 : MC_ReadActualVelocity; (*Function Block *)
	MC_ReadStatus_0 : MC_ReadStatus; (*Function Block *)
	MC_Stop_0 : MC_Stop; (*Function Block *)
END_VAR
```
